  MoveL 2054 to (540.62, 2920.87, 513.19) mm, rotated rx -180 ry 0 rz -88.32 deg; joints [12.318, 40.901, 21.897, 21.013, -28.48, -28.65]
  MoveL 2055 to (543.06, 2922.34, 513.19) mm, rotated rx 180 ry 0 rz -88.32 deg; joints [12.364, 41.01, 22.057, 21.039, -28.543, -28.697]
  MoveL 2056 to (545.51, 2923.81, 513.19) mm, rotated rx -180 ry 0 rz -88.32 deg; joints [12.409, 41.12, 22.218, 21.064, -28.606, -28.743]
  MoveL 2057 to (547.96, 2925.26, 513.19) mm, rotated rx -180 ry 0 rz -88.32 deg; joints [12.455, 41.229, 22.379, 21.09, -28.67, -28.789]
  MoveL 2058 to (550.41, 2926.72, 513.19) mm, rotated rx 180 ry 0 rz -88.32 deg; joints [12.501, 41.339, 22.539, 21.115, -28.733, -28.835]
  MoveL 2059 to (552.87, 2928.16, 513.19) mm, rotated rx -180 ry 0 rz -88.32 deg; joints [12.547, 41.448, 22.7, 21.141, -28.797, -28.881]
  MoveL 2060 to (555.33, 2929.6, 513.19) mm, rotated rx -180 ry 0 rz -88.32 deg; joints [12.593, 41.558, 22.861, 21.166, -28.86, -28.926]
  MoveL 2061 to (557.79, 2931.02, 513.19) mm, rotated rx 180 ry 0 rz -88.32 deg; joints [12.639, 41.667, 23.021, 21.191, -28.924, -28.972]
  MoveL 2062 to (560.26, 2932.45, 513.19) mm, rotated rx 180 ry 0 rz -88.32 deg; joints [12.685, 41.776, 23.182, 21.216, -28.988, -29.018]
  MoveL 2063 to (562.74, 2933.86, 513.19) mm, rotated rx -180 ry 0 rz -88.32 deg; joints [12.731, 41.885, 23.343, 21.241, -29.052, -29.063]
  MoveL 2064 to (565.21, 2935.27, 513.19) mm, rotated rx -180 ry 0 rz -88.32 deg; joints [12.777, 41.995, 23.504, 21.266, -29.116, -29.108]
  MoveL 2065 to (567.69, 2936.67, 513.19) mm, rotated rx -180 ry 0 rz -88.32 deg; joints [12.823, 42.104, 23.665, 21.291, -29.18, -29.154]
  MoveL 2066 to (570.18, 2938.07, 513.19) mm, rotated rx 180 ry 0 rz -88.32 deg; joints [12.87, 42.213, 23.826, 21.316, -29.244, -29.199]
  MoveL 2067 to (572.67, 2939.46, 513.19) mm, rotated rx 180 ry 0 rz -88.32 deg; joints [12.916, 42.322, 23.987, 21.341, -29.309, -29.244]
  MoveL 2068 to (575.16, 2940.84, 513.19) mm, rotated rx 180 ry 0 rz -88.32 deg; joints [12.962, 42.431, 24.148, 21.366, -29.373, -29.289]
  MoveL 2069 to (577.66, 2942.21, 513.19) mm, rotated rx 180 ry 0 rz -88.32 deg; joints [13.009, 42.54, 24.31, 21.39, -29.438, -29.334]
  MoveL 2070 to (580.16, 2943.58, 513.19) mm, rotated rx 180 ry 0 rz -88.32 deg; joints [13.055, 42.649, 24.471, 21.415, -29.502, -29.378]
  MoveL 2071 to (582.66, 2944.94, 513.19) mm, rotated rx 180 ry 0 rz -88.32 deg; joints [13.102, 42.758, 24.632, 21.439, -29.567, -29.423]
  MoveL 2072 to (585.17, 2946.29, 513.19) mm, rotated rx 180 ry 0 rz -88.32 deg; joints [13.148, 42.867, 24.793, 21.463, -29.632, -29.468]
  MoveL 2073 to (587.68, 2947.64, 513.19) mm, rotated rx -180 ry 0 rz -88.32 deg; joints [13.195, 42.976, 24.955, 21.487, -29.697, -29.512]
  MoveL 2074 to (590.2, 2948.98, 513.19) mm, rotated rx -180 ry 0 rz -88.32 deg; joints [13.241, 43.085, 25.116, 21.512, -29.762, -29.557]
  MoveL 2075 to (592.72, 2950.31, 513.19) mm, rotated rx -180 ry 0 rz -88.32 deg; joints [13.288, 43.194, 25.278, 21.536, -29.828, -29.601]
  MoveL 2076 to (595.24, 2951.63, 513.19) mm, rotated rx -180 ry 0 rz -88.32 deg; joints [13.335, 43.303, 25.439, 21.56, -29.893, -29.645]
  MoveL 2077 to (597.77, 2952.95, 513.19) mm, rotated rx -180 ry 0 rz -88.32 deg; joints [13.382, 43.412, 25.601, 21.584, -29.959, -29.689]
  MoveL 2078 to (600.3, 2954.26, 513.19) mm, rotated rx 180 ry 0 rz -88.32 deg; joints [13.429, 43.521, 25.763, 21.607, -30.024, -29.733]
  MoveL 2079 to (602.83, 2955.57, 513.19) mm, rotated rx 180 ry 0 rz -88.32 deg; joints [13.475, 43.629, 25.924, 21.631, -30.09, -29.777]
  MoveL 2080 to (605.37, 2956.86, 513.19) mm, rotated rx 180 ry 0 rz -88.32 deg; joints [13.522, 43.738, 26.086, 21.655, -30.156, -29.821]
  MoveL 2081 to (607.91, 2958.15, 513.19) mm, rotated rx -180 ry 0 rz -88.32 deg; joints [13.569, 43.847, 26.248, 21.678, -30.222, -29.865]
  MoveL 2082 to (610.46, 2959.43, 513.19) mm, rotated rx -180 ry 0 rz -88.32 deg; joints [13.616, 43.955, 26.41, 21.702, -30.288, -29.908]
  MoveL 2083 to (613.01, 2960.71, 513.19) mm, rotated rx -180 ry 0 rz -88.32 deg; joints [13.663, 44.064, 26.572, 21.725, -30.354, -29.952]
  MoveL 2084 to (615.56, 2961.98, 513.19) mm, rotated rx 180 ry 0 rz -88.32 deg; joints [13.711, 44.173, 26.734, 21.749, -30.42, -29.996]
  MoveL 2085 to (618.11, 2963.24, 513.19) mm, rotated rx -180 ry 0 rz -88.32 deg; joints [13.758, 44.281, 26.896, 21.772, -30.486, -30.039]
  MoveL 2086 to (620.67, 2964.49, 513.19) mm, rotated rx 180 ry 0 rz -88.32 deg; joints [13.805, 44.39, 27.058, 21.795, -30.553, -30.082]
  MoveL 2087 to (623.24, 2965.74, 513.19) mm, rotated rx -180 ry 0 rz -88.32 deg; joints [13.852, 44.498, 27.22, 21.818, -30.619, -30.125]
  MoveL 2088 to (625.8, 2966.98, 513.19) mm, rotated rx -180 ry 0 rz -88.32 deg; joints [13.899, 44.607, 27.383, 21.841, -30.686, -30.168]
  MoveL 2089 to (628.37, 2968.21, 513.19) mm, rotated rx -180 ry 0 rz -88.32 deg; joints [13.947, 44.715, 27.545, 21.864, -30.753, -30.211]
  MoveL 2090 to (630.95, 2969.43, 513.19) mm, rotated rx -180 ry 0 rz -88.32 deg; joints [13.994, 44.824, 27.707, 21.887, -30.82, -30.254]
  MoveL 2091 to (633.52, 2970.65, 513.19) mm, rotated rx 180 ry 0 rz -88.32 deg; joints [14.042, 44.932, 27.87, 21.91, -30.887, -30.297]
  MoveL 2092 to (636.1, 2971.86, 513.19) mm, rotated rx -180 ry 0 rz -88.32 deg; joints [14.089, 45.041, 28.032, 21.933, -30.954, -30.34]
  MoveL 2093 to (638.69, 2973.06, 513.19) mm, rotated rx -180 ry 0 rz -88.32 deg; joints [14.137, 45.149, 28.195, 21.955, -31.021, -30.382]
  MoveL 2094 to (641.27, 2974.26, 513.19) mm, rotated rx 180 ry 0 rz -88.32 deg; joints [14.184, 45.257, 28.357, 21.978, -31.088, -30.425]
  MoveL 2095 to (643.86, 2975.45, 513.19) mm, rotated rx -180 ry 0 rz -88.32 deg; joints [14.232, 45.366, 28.52, 22, -31.156, -30.467]
  MoveL 2096 to (646.46, 2976.63, 513.19) mm, rotated rx 180 ry 0 rz -88.32 deg; joints [14.28, 45.474, 28.682, 22.023, -31.223, -30.51]
  MoveL 2097 to (649.05, 2977.8, 513.19) mm, rotated rx -180 ry 0 rz -88.32 deg; joints [14.327, 45.582, 28.845, 22.045, -31.291, -30.552]
  MoveL 2098 to (651.65, 2978.97, 513.19) mm, rotated rx -180 ry 0 rz -88.32 deg; joints [14.375, 45.691, 29.008, 22.067, -31.358, -30.594]
  MoveL 2099 to (654.26, 2980.13, 513.19) mm, rotated rx 180 ry 0 rz -88.32 deg; joints [14.423, 45.799, 29.171, 22.089, -31.426, -30.636]
  MoveL 2100 to (656.86, 2981.28, 513.19) mm, rotated rx 180 ry 0 rz -88.32 deg; joints [14.471, 45.907, 29.334, 22.112, -31.494, -30.678]
  MoveL 2101 to (659.47, 2982.43, 513.19) mm, rotated rx -180 ry 0 rz -88.32 deg; joints [14.518, 46.015, 29.497, 22.134, -31.562, -30.72]
  MoveL 2102 to (662.09, 2983.56, 513.19) mm, rotated rx -180 ry 0 rz -88.32 deg; joints [14.566, 46.124, 29.66, 22.156, -31.63, -30.762]
  MoveL 2103 to (664.7, 2984.69, 513.19) mm, rotated rx -180 ry 0 rz -88.32 deg; joints [14.614, 46.232, 29.823, 22.177, -31.699, -30.803]
  MoveL 2104 to (667.32, 2985.82, 513.19) mm, rotated rx 180 ry 0 rz -88.32 deg; joints [14.662, 46.34, 29.986, 22.199, -31.767, -30.845]
  MoveL 2105 to (669.95, 2986.93, 513.19) mm, rotated rx -180 ry 0 rz -88.32 deg; joints [14.71, 46.448, 30.149, 22.221, -31.835, -30.886]
  MoveL 2106 to (672.57, 2988.04, 513.19) mm, rotated rx 180 ry 0 rz -88.32 deg; joints [14.759, 46.556, 30.313, 22.243, -31.904, -30.928]
  MoveL 2107 to (675.2, 2989.14, 513.19) mm, rotated rx -180 ry 0 rz -88.32 deg; joints [14.807, 46.664, 30.476, 22.264, -31.973, -30.969]
  MoveL 2108 to (677.83, 2990.23, 513.19) mm, rotated rx -180 ry 0 rz -88.32 deg; joints [14.855, 46.772, 30.64, 22.286, -32.041, -31.01]
  MoveL 2109 to (680.47, 2991.32, 513.19) mm, rotated rx 180 ry 0 rz -88.32 deg; joints [14.903, 46.88, 30.803, 22.307, -32.11, -31.051]
  MoveL 2110 to (683.1, 2992.4, 513.19) mm, rotated rx 180 ry 0 rz -88.32 deg; joints [14.951, 46.988, 30.967, 22.329, -32.179, -31.092]
  MoveL 2111 to (685.75, 2993.47, 513.19) mm, rotated rx -180 ry 0 rz -88.32 deg; joints [15, 47.097, 31.13, 22.35, -32.248, -31.133]
  MoveL 2112 to (688.39, 2994.53, 513.19) mm, rotated rx 180 ry 0 rz -88.32 deg; joints [15.048, 47.205, 31.294, 22.371, -32.317, -31.174]
  MoveL 2113 to (691.04, 2995.59, 513.19) mm, rotated rx 180 ry 0 rz -88.32 deg; joints [15.096, 47.313, 31.458, 22.392, -32.387, -31.215]
  MoveL 2114 to (693.69, 2996.64, 513.19) mm, rotated rx -180 ry 0 rz -88.32 deg; joints [15.145, 47.421, 31.622, 22.413, -32.456, -31.255]
  MoveL 2115 to (696.34, 2997.68, 513.19) mm, rotated rx 180 ry 0 rz -88.32 deg; joints [15.193, 47.528, 31.786, 22.434, -32.526, -31.296]
  MoveL 2116 to (698.99, 2998.71, 513.19) mm, rotated rx 180 ry 0 rz -88.32 deg; joints [15.242, 47.636, 31.949, 22.455, -32.595, -31.336]
  MoveL 2117 to (701.65, 2999.74, 513.19) mm, rotated rx -180 ry 0 rz -88.32 deg; joints [15.29, 47.744, 32.114, 22.476, -32.665, -31.377]
  MoveL 2118 to (704.31, 3000.76, 513.19) mm, rotated rx -180 ry 0 rz -88.32 deg; joints [15.339, 47.852, 32.278, 22.497, -32.735, -31.417]
  MoveL 2119 to (706.98, 3001.77, 513.19) mm, rotated rx -180 ry 0 rz -88.32 deg; joints [15.387, 47.96, 32.442, 22.518, -32.805, -31.457]
  MoveL 2120 to (709.65, 3002.77, 513.19) mm, rotated rx -180 ry 0 rz -88.32 deg; joints [15.436, 48.068, 32.606, 22.538, -32.875, -31.497]
  MoveL 2121 to (712.32, 3003.77, 513.19) mm, rotated rx 180 ry 0 rz -88.32 deg; joints [15.485, 48.176, 32.77, 22.559, -32.945, -31.537]
  MoveL 2122 to (714.99, 3004.76, 513.19) mm, rotated rx 180 ry 0 rz -88.32 deg; joints [15.533, 48.284, 32.935, 22.58, -33.015, -31.577]
  MoveL 2123 to (717.66, 3005.74, 513.19) mm, rotated rx 180 ry 0 rz -88.32 deg; joints [15.582, 48.392, 33.099, 22.6, -33.085, -31.617]
  MoveL 2124 to (720.34, 3006.71, 513.19) mm, rotated rx -180 ry 0 rz -88.32 deg; joints [15.631, 48.5, 33.264, 22.62, -33.156, -31.656]
  MoveL 2125 to (723.02, 3007.68, 513.19) mm, rotated rx -180 ry 0 rz -88.32 deg; joints [15.68, 48.607, 33.428, 22.641, -33.226, -31.696]
  MoveL 2126 to (725.71, 3008.64, 513.19) mm, rotated rx 180 ry 0 rz -88.32 deg; joints [15.729, 48.715, 33.593, 22.661, -33.297, -31.735]
  MoveL 2127 to (728.39, 3009.59, 513.19) mm, rotated rx 180 ry 0 rz -88.32 deg; joints [15.778, 48.823, 33.758, 22.681, -33.368, -31.775]
  MoveL 2128 to (731.08, 3010.54, 513.19) mm, rotated rx -180 ry 0 rz -88.32 deg; joints [15.827, 48.931, 33.923, 22.701, -33.438, -31.814]
  MoveL 2129 to (733.77, 3011.47, 513.19) mm, rotated rx -180 ry 0 rz -88.32 deg; joints [15.876, 49.039, 34.087, 22.721, -33.509, -31.853]
  MoveL 2130 to (736.47, 3012.4, 513.19) mm, rotated rx 180 ry 0 rz -88.32 deg; joints [15.925, 49.147, 34.252, 22.741, -33.58, -31.892]
  MoveL 2131 to (739.16, 3013.32, 513.19) mm, rotated rx -180 ry 0 rz -88.32 deg; joints [15.974, 49.254, 34.417, 22.761, -33.651, -31.931]
  MoveL 2132 to (741.86, 3014.24, 513.19) mm, rotated rx -180 ry 0 rz -88.32 deg; joints [16.023, 49.362, 34.583, 22.781, -33.723, -31.97]
  MoveL 2133 to (744.57, 3015.14, 513.19) mm, rotated rx -180 ry 0 rz -88.32 deg; joints [16.072, 49.47, 34.748, 22.801, -33.794, -32.009]
  MoveL 2134 to (747.27, 3016.04, 513.19) mm, rotated rx 180 ry 0 rz -88.32 deg; joints [16.121, 49.578, 34.913, 22.821, -33.865, -32.048]
  MoveL 2135 to (749.98, 3016.93, 513.19) mm, rotated rx 180 ry 0 rz -88.32 deg; joints [16.17, 49.686, 35.078, 22.84, -33.937, -32.087]
  MoveL 2136 to (752.69, 3017.82, 513.19) mm, rotated rx -180 ry 0 rz -88.32 deg; joints [16.22, 49.793, 35.244, 22.86, -34.009, -32.125]
  MoveL 2137 to (755.4, 3018.69, 513.19) mm, rotated rx -180 ry 0 rz -88.32 deg; joints [16.269, 49.901, 35.409, 22.879, -34.08, -32.164]
  MoveL 2138 to (758.11, 3019.56, 513.19) mm, rotated rx -180 ry 0 rz -88.32 deg; joints [16.318, 50.009, 35.575, 22.899, -34.152, -32.202]
  MoveL 2139 to (760.83, 3020.42, 513.19) mm, rotated rx -180 ry 0 rz -88.32 deg; joints [16.368, 50.117, 35.741, 22.918, -34.224, -32.24]
  MoveL 2140 to (763.55, 3021.27, 513.19) mm, rotated rx 180 ry 0 rz -88.32 deg; joints [16.417, 50.224, 35.906, 22.937, -34.296, -32.278]
  MoveL 2141 to (766.27, 3022.12, 513.19) mm, rotated rx -180 ry 0 rz -88.32 deg; joints [16.466, 50.332, 36.072, 22.957, -34.368, -32.316]
  MoveL 2142 to (769, 3022.96, 513.19) mm, rotated rx -180 ry 0 rz -88.32 deg; joints [16.516, 50.44, 36.238, 22.976, -34.441, -32.354]
  MoveL 2143 to (771.72, 3023.79, 513.19) mm, rotated rx 180 ry 0 rz -88.32 deg; joints [16.565, 50.548, 36.404, 22.995, -34.513, -32.392]
  MoveL 2144 to (774.45, 3024.61, 513.19) mm, rotated rx -180 ry 0 rz -88.32 deg; joints [16.615, 50.655, 36.57, 23.014, -34.585, -32.43]
  MoveL 2145 to (777.18, 3025.42, 513.19) mm, rotated rx 180 ry 0 rz -88.32 deg; joints [16.665, 50.763, 36.736, 23.033, -34.658, -32.468]
  MoveL 2146 to (779.91, 3026.23, 513.19) mm, rotated rx 180 ry 0 rz -88.32 deg; joints [16.714, 50.871, 36.903, 23.052, -34.731, -32.505]
  MoveL 2147 to (782.65, 3027.03, 513.19) mm, rotated rx -180 ry 0 rz -88.32 deg; joints [16.764, 50.979, 37.069, 23.071, -34.803, -32.543]
  MoveL 2148 to (785.39, 3027.82, 513.19) mm, rotated rx -180 ry 0 rz -88.32 deg; joints [16.814, 51.086, 37.235, 23.09, -34.876, -32.58]
  MoveL 2149 to (788.13, 3028.61, 513.19) mm, rotated rx -180 ry 0 rz -88.32 deg; joints [16.863, 51.194, 37.402, 23.108, -34.949, -32.618]
  MoveL 2150 to (790.87, 3029.38, 513.19) mm, rotated rx -180 ry 0 rz -88.32 deg; joints [16.913, 51.302, 37.568, 23.127, -35.022, -32.655]
  MoveL 2151 to (793.61, 3030.15, 513.19) mm, rotated rx -180 ry 0 rz -88.32 deg; joints [16.963, 51.41, 37.735, 23.145, -35.095, -32.692]
  MoveL 2152 to (796.36, 3030.91, 513.19) mm, rotated rx 180 ry 0 rz -88.32 deg; joints [17.013, 51.518, 37.902, 23.164, -35.169, -32.729]
  MoveL 2153 to (799.11, 3031.66, 513.19) mm, rotated rx -180 ry 0 rz -88.32 deg; joints [17.062, 51.625, 38.069, 23.183, -35.242, -32.766]
  MoveL 2154 to (801.86, 3032.41, 513.19) mm, rotated rx -180 ry 0 rz -88.32 deg; joints [17.112, 51.733, 38.236, 23.201, -35.316, -32.803]
  MoveL 2155 to (804.61, 3033.15, 513.19) mm, rotated rx 180 ry 0 rz -88.32 deg; joints [17.162, 51.841, 38.403, 23.219, -35.389, -32.84]
  MoveL 2156 to (807.37, 3033.88, 513.19) mm, rotated rx 180 ry 0 rz -88.32 deg; joints [17.212, 51.949, 38.57, 23.238, -35.463, -32.876]
  MoveL 2157 to (810.12, 3034.6, 513.19) mm, rotated rx 180 ry 0 rz -88.32 deg; joints [17.262, 52.057, 38.737, 23.256, -35.537, -32.913]
  MoveL 2158 to (812.88, 3035.31, 513.19) mm, rotated rx -180 ry 0 rz -88.32 deg; joints [17.312, 52.164, 38.904, 23.274, -35.611, -32.949]
  MoveL 2159 to (815.64, 3036.02, 513.19) mm, rotated rx -180 ry 0 rz -88.32 deg; joints [17.362, 52.272, 39.072, 23.292, -35.685, -32.986]
  MoveL 2160 to (818.41, 3036.72, 513.19) mm, rotated rx 180 ry 0 rz -88.32 deg; joints [17.412, 52.38, 39.239, 23.31, -35.759, -33.022]
  MoveL 2161 to (821.17, 3037.41, 513.19) mm, rotated rx 180 ry 0 rz -88.32 deg; joints [17.462, 52.488, 39.407, 23.328, -35.833, -33.058]
  MoveL 2162 to (823.94, 3038.1, 513.19) mm, rotated rx -180 ry 0 rz -88.32 deg; joints [17.513, 52.596, 39.575, 23.346, -35.907, -33.094]
  MoveL 2163 to (826.71, 3038.77, 513.19) mm, rotated rx -180 ry 0 rz -88.32 deg; joints [17.563, 52.704, 39.743, 23.364, -35.982, -33.13]
  MoveL 2164 to (829.48, 3039.44, 513.19) mm, rotated rx 180 ry 0 rz -88.32 deg; joints [17.613, 52.812, 39.911, 23.382, -36.056, -33.166]
  MoveL 2165 to (832.25, 3040.1, 513.19) mm, rotated rx 180 ry 0 rz -88.32 deg; joints [17.663, 52.919, 40.079, 23.399, -36.131, -33.202]
  MoveL 2166 to (835.02, 3040.75, 513.19) mm, rotated rx -180 ry 0 rz -88.32 deg; joints [17.714, 53.027, 40.247, 23.417, -36.206, -33.238]
  MoveL 2167 to (837.8, 3041.4, 513.19) mm, rotated rx 180 ry 0 rz -88.32 deg; joints [17.764, 53.135, 40.415, 23.435, -36.28, -33.273]
  MoveL 2168 to (840.58, 3042.03, 513.19) mm, rotated rx 180 ry 0 rz -88.32 deg; joints [17.814, 53.243, 40.583, 23.452, -36.355, -33.309]
  MoveL 2169 to (843.36, 3042.66, 513.19) mm, rotated rx -180 ry 0 rz -88.32 deg; joints [17.865, 53.351, 40.752, 23.47, -36.43, -33.344]
  MoveL 2170 to (846.14, 3043.28, 513.19) mm, rotated rx 180 ry 0 rz -88.32 deg; joints [17.915, 53.459, 40.92, 23.487, -36.506, -33.379]
  MoveL 2171 to (848.92, 3043.9, 513.19) mm, rotated rx -180 ry 0 rz -88.32 deg; joints [17.965, 53.567, 41.089, 23.505, -36.581, -33.415]
  MoveL 2172 to (851.7, 3044.5, 513.19) mm, rotated rx -180 ry 0 rz -88.32 deg; joints [18.016, 53.675, 41.258, 23.522, -36.656, -33.45]
  MoveL 2173 to (854.49, 3045.1, 513.19) mm, rotated rx 180 ry 0 rz -88.32 deg; joints [18.066, 53.783, 41.427, 23.539, -36.732, -33.485]
  MoveL 2174 to (857.28, 3045.69, 513.19) mm, rotated rx 180 ry 0 rz -88.32 deg; joints [18.117, 53.891, 41.596, 23.556, -36.807, -33.52]
  MoveL 2175 to (860.07, 3046.27, 513.19) mm, rotated rx -180 ry 0 rz -88.32 deg; joints [18.167, 54, 41.765, 23.573, -36.883, -33.555]
  MoveL 2176 to (862.86, 3046.85, 513.19) mm, rotated rx 180 ry 0 rz -88.32 deg; joints [18.218, 54.108, 41.934, 23.59, -36.959, -33.589]
  MoveL 2177 to (865.65, 3047.42, 513.19) mm, rotated rx 180 ry 0 rz -88.32 deg; joints [18.269, 54.216, 42.103, 23.607, -37.035, -33.624]
  MoveL 2178 to (868.45, 3047.97, 513.19) mm, rotated rx -180 ry 0 rz -88.32 deg; joints [18.319, 54.324, 42.273, 23.624, -37.111, -33.659]
  MoveL 2179 to (871.24, 3048.53, 513.19) mm, rotated rx 180 ry 0 rz -88.32 deg; joints [18.37, 54.432, 42.442, 23.641, -37.187, -33.693]
  MoveL 2180 to (874.04, 3049.07, 513.19) mm, rotated rx 180 ry 0 rz -88.32 deg; joints [18.421, 54.54, 42.612, 23.658, -37.263, -33.727]
  MoveL 2181 to (876.84, 3049.6, 513.19) mm, rotated rx 180 ry 0 rz -88.32 deg; joints [18.471, 54.649, 42.782, 23.675, -37.339, -33.762]
  MoveL 2182 to (879.64, 3050.13, 513.19) mm, rotated rx 180 ry 0 rz -88.32 deg; joints [18.522, 54.757, 42.952, 23.692, -37.416, -33.796]
  MoveL 2183 to (882.44, 3050.65, 513.19) mm, rotated rx 180 ry 0 rz -88.32 deg; joints [18.573, 54.865, 43.122, 23.708, -37.492, -33.83]
  MoveL 2184 to (885.25, 3051.16, 513.19) mm, rotated rx -180 ry 0 rz -88.32 deg; joints [18.624, 54.974, 43.292, 23.725, -37.569, -33.864]
  MoveL 2185 to (888.05, 3051.67, 513.19) mm, rotated rx 180 ry 0 rz -88.32 deg; joints [18.675, 55.082, 43.463, 23.741, -37.646, -33.897]
  MoveL 2186 to (890.86, 3052.16, 513.19) mm, rotated rx 180 ry 0 rz -88.32 deg; joints [18.726, 55.19, 43.633, 23.758, -37.723, -33.931]
  MoveL 2187 to (893.67, 3052.65, 513.19) mm, rotated rx -180 ry 0 rz -88.32 deg; joints [18.776, 55.299, 43.804, 23.774, -37.8, -33.965]
  MoveL 2188 to (896.48, 3053.13, 513.19) mm, rotated rx 180 ry 0 rz -88.32 deg; joints [18.827, 55.407, 43.974, 23.791, -37.877, -33.998]
  MoveL 2189 to (899.29, 3053.6, 513.19) mm, rotated rx -180 ry 0 rz -88.32 deg; joints [18.878, 55.516, 44.145, 23.807, -37.954, -34.032]
  MoveL 2190 to (902.1, 3054.07, 513.19) mm, rotated rx -180 ry 0 rz -88.32 deg; joints [18.929, 55.624, 44.316, 23.823, -38.031, -34.065]
  MoveL 2191 to (904.91, 3054.52, 513.19) mm, rotated rx -180 ry 0 rz -88.32 deg; joints [18.98, 55.733, 44.487, 23.839, -38.109, -34.098]
  MoveL 2192 to (907.72, 3054.97, 513.19) mm, rotated rx 180 ry 0 rz -88.32 deg; joints [19.031, 55.842, 44.659, 23.856, -38.186, -34.132]
  MoveL 2193 to (910.54, 3055.41, 513.19) mm, rotated rx -180 ry 0 rz -88.32 deg; joints [19.082, 55.95, 44.83, 23.872, -38.264, -34.165]
  MoveL 2194 to (913.36, 3055.85, 513.19) mm, rotated rx -180 ry 0 rz -88.32 deg; joints [19.134, 56.059, 45.002, 23.888, -38.342, -34.198]
  MoveL 2195 to (916.18, 3056.27, 513.19) mm, rotated rx 180 ry 0 rz -88.32 deg; joints [19.185, 56.168, 45.173, 23.904, -38.419, -34.23]
  MoveL 2196 to (918.99, 3056.69, 513.19) mm, rotated rx -180 ry 0 rz -88.32 deg; joints [19.236, 56.276, 45.345, 23.92, -38.497, -34.263]
  MoveL 2197 to (921.81, 3057.1, 513.19) mm, rotated rx 180 ry 0 rz -88.32 deg; joints [19.287, 56.385, 45.517, 23.935, -38.576, -34.296]
  MoveL 2198 to (924.64, 3057.5, 513.19) mm, rotated rx -180 ry 0 rz -88.32 deg; joints [19.338, 56.494, 45.689, 23.951, -38.654, -34.328]
  MoveL 2199 to (927.46, 3057.89, 513.19) mm, rotated rx -180 ry 0 rz -88.32 deg; joints [19.39, 56.603, 45.862, 23.967, -38.732, -34.361]
  MoveL 2200 to (930.28, 3058.28, 513.19) mm, rotated rx -180 ry 0 rz -88.32 deg; joints [19.441, 56.712, 46.034, 23.983, -38.811, -34.393]
  MoveL 2201 to (933.11, 3058.65, 513.19) mm, rotated rx -180 ry 0 rz -88.32 deg; joints [19.492, 56.821, 46.207, 23.998, -38.889, -34.425]
  MoveL 2202 to (935.93, 3059.02, 513.19) mm, rotated rx -180 ry 0 rz -88.32 deg; joints [19.543, 56.93, 46.379, 24.014, -38.968, -34.457]
  MoveL 2203 to (938.76, 3059.39, 513.19) mm, rotated rx -180 ry 0 rz -88.32 deg; joints [19.595, 57.039, 46.552, 24.029, -39.047, -34.489]
  MoveL 2204 to (941.59, 3059.74, 513.19) mm, rotated rx -180 ry 0 rz -88.32 deg; joints [19.646, 57.149, 46.725, 24.045, -39.126, -34.521]
  MoveL 2205 to (944.42, 3060.09, 513.19) mm, rotated rx 180 ry 0 rz -88.32 deg; joints [19.698, 57.258, 46.899, 24.06, -39.205, -34.553]
  MoveL 2206 to (947.25, 3060.42, 513.19) mm, rotated rx -180 ry 0 rz -88.32 deg; joints [19.749, 57.367, 47.072, 24.075, -39.284, -34.585]
  MoveL 2207 to (950.08, 3060.75, 513.19) mm, rotated rx -180 ry 0 rz -88.32 deg; joints [19.8, 57.477, 47.246, 24.091, -39.363, -34.616]
  MoveL 2208 to (952.91, 3061.07, 513.19) mm, rotated rx 180 ry 0 rz -88.32 deg; joints [19.852, 57.586, 47.42, 24.106, -39.443, -34.648]
  MoveL 2209 to (955.74, 3061.39, 513.19) mm, rotated rx -180 ry 0 rz -88.32 deg; joints [19.903, 57.695, 47.593, 24.121, -39.522, -34.679]
  MoveL 2210 to (958.57, 3061.7, 513.19) mm, rotated rx -180 ry 0 rz -88.32 deg; joints [19.955, 57.805, 47.768, 24.136, -39.602, -34.71]
  MoveL 2211 to (961.41, 3061.99, 513.19) mm, rotated rx 180 ry 0 rz -88.32 deg; joints [20.006, 57.915, 47.942, 24.151, -39.682, -34.742]
  MoveL 2212 to (964.24, 3062.28, 513.19) mm, rotated rx 180 ry 0 rz -88.32 deg; joints [20.058, 58.024, 48.116, 24.166, -39.762, -34.773]
  MoveL 2213 to (967.08, 3062.57, 513.19) mm, rotated rx -180 ry 0 rz -88.32 deg; joints [20.11, 58.134, 48.291, 24.181, -39.842, -34.804]
  MoveL 2214 to (969.92, 3062.84, 513.19) mm, rotated rx -180 ry 0 rz -88.32 deg; joints [20.161, 58.244, 48.466, 24.196, -39.922, -34.834]
  MoveL 2215 to (972.75, 3063.11, 513.19) mm, rotated rx 180 ry 0 rz -88.32 deg; joints [20.213, 58.354, 48.641, 24.211, -40.002, -34.865]
  MoveL 2216 to (975.59, 3063.36, 513.19) mm, rotated rx 180 ry 0 rz -88.32 deg; joints [20.265, 58.464, 48.816, 24.225, -40.082, -34.896]
  MoveL 2217 to (978.43, 3063.61, 513.19) mm, rotated rx -180 ry 0 rz -88.32 deg; joints [20.316, 58.574, 48.992, 24.24, -40.163, -34.926]
  MoveL 2218 to (981.27, 3063.86, 513.19) mm, rotated rx -180 ry 0 rz -88.32 deg; joints [20.368, 58.684, 49.167, 24.255, -40.244, -34.957]
  MoveL 2219 to (984.11, 3064.09, 513.19) mm, rotated rx -180 ry 0 rz -88.32 deg; joints [20.42, 58.794, 49.343, 24.269, -40.324, -34.987]
  MoveL 2220 to (986.95, 3064.32, 513.19) mm, rotated rx 180 ry 0 rz -88.32 deg; joints [20.472, 58.904, 49.519, 24.284, -40.405, -35.017]
  MoveL 2221 to (989.79, 3064.54, 513.19) mm, rotated rx -180 ry 0 rz -88.32 deg; joints [20.523, 59.015, 49.695, 24.298, -40.486, -35.047]
  MoveL 2222 to (992.63, 3064.75, 513.19) mm, rotated rx 180 ry 0 rz -88.32 deg; joints [20.575, 59.125, 49.872, 24.313, -40.568, -35.077]
  MoveL 2223 to (995.48, 3064.95, 513.19) mm, rotated rx -180 ry 0 rz -88.32 deg; joints [20.627, 59.236, 50.049, 24.327, -40.649, -35.107]
  MoveL 2224 to (998.32, 3065.14, 513.19) mm, rotated rx 180 ry 0 rz -88.32 deg; joints [20.679, 59.347, 50.225, 24.341, -40.73, -35.136]
  MoveL 2225 to (1001.16, 3065.33, 513.19) mm, rotated rx -180 ry 0 rz -88.32 deg; joints [20.731, 59.457, 50.403, 24.355, -40.812, -35.166]
  MoveL 2226 to (1004.01, 3065.51, 513.19) mm, rotated rx 180 ry 0 rz -88.32 deg; joints [20.783, 59.568, 50.58, 24.37, -40.894, -35.196]
  MoveL 2227 to (1006.85, 3065.68, 513.19) mm, rotated rx -180 ry 0 rz -88.32 deg; joints [20.835, 59.679, 50.757, 24.384, -40.976, -35.225]
  MoveL 2228 to (1009.7, 3065.84, 513.19) mm, rotated rx 180 ry 0 rz -88.32 deg; joints [20.887, 59.79, 50.935, 24.398, -41.058, -35.254]
  MoveL 2229 to (1012.54, 3066, 513.19) mm, rotated rx -180 ry 0 rz -88.32 deg; joints [20.939, 59.901, 51.113, 24.412, -41.14, -35.283]
  MoveL 2230 to (1015.39, 3066.14, 513.19) mm, rotated rx -180 ry 0 rz -88.32 deg; joints [20.991, 60.012, 51.292, 24.426, -41.222, -35.312]
  MoveL 2231 to (1018.24, 3066.28, 513.19) mm, rotated rx -180 ry 0 rz -88.32 deg; joints [21.043, 60.124, 51.47, 24.439, -41.305, -35.341]
  MoveL 2232 to (1021.08, 3066.41, 513.19) mm, rotated rx -180 ry 0 rz -88.32 deg; joints [21.095, 60.235, 51.649, 24.453, -41.387, -35.37]
  MoveL 2233 to (1023.93, 3066.54, 513.19) mm, rotated rx 180 ry 0 rz -88.32 deg; joints [21.147, 60.347, 51.828, 24.467, -41.47, -35.398]
  MoveL 2234 to (1026.78, 3066.65, 513.19) mm, rotated rx -180 ry 0 rz -88.32 deg; joints [21.199, 60.458, 52.007, 24.481, -41.553, -35.427]
  MoveL 2235 to (1029.63, 3066.76, 513.19) mm, rotated rx -180 ry 0 rz -88.32 deg; joints [21.251, 60.57, 52.187, 24.494, -41.636, -35.455]
  MoveL 2236 to (1032.47, 3066.86, 513.19) mm, rotated rx -180 ry 0 rz -88.32 deg; joints [21.303, 60.682, 52.367, 24.508, -41.719, -35.484]
  MoveL 2237 to (1035.32, 3066.95, 513.19) mm, rotated rx -180 ry 0 rz -88.32 deg; joints [21.355, 60.794, 52.547, 24.521, -41.802, -35.512]
  MoveL 2238 to (1038.17, 3067.03, 513.19) mm, rotated rx 180 ry 0 rz -88.32 deg; joints [21.407, 60.906, 52.727, 24.535, -41.886, -35.54]
  MoveL 2239 to (1041.02, 3067.11, 513.19) mm, rotated rx -180 ry 0 rz -88.32 deg; joints [21.46, 61.019, 52.908, 24.548, -41.969, -35.568]
  MoveL 2240 to (1043.87, 3067.17, 513.19) mm, rotated rx -180 ry 0 rz -88.32 deg; joints [21.512, 61.131, 53.089, 24.561, -42.053, -35.595]
  MoveL 2241 to (1046.72, 3067.23, 513.19) mm, rotated rx 180 ry 0 rz -88.32 deg; joints [21.564, 61.244, 53.27, 24.574, -42.137, -35.623]
  MoveL 2242 to (1049.57, 3067.28, 513.19) mm, rotated rx -180 ry 0 rz -88.32 deg; joints [21.616, 61.356, 53.451, 24.587, -42.221, -35.65]
  MoveL 2243 to (1052.42, 3067.32, 513.19) mm, rotated rx -180 ry 0 rz -88.32 deg; joints [21.669, 61.469, 53.633, 24.601, -42.306, -35.678]
  MoveL 2244 to (1055.27, 3067.36, 513.19) mm, rotated rx -180 ry 0 rz -88.32 deg; joints [21.721, 61.582, 53.815, 24.614, -42.39, -35.705]
  MoveL 2245 to (1058.12, 3067.39, 513.19) mm, rotated rx -180 ry 0 rz -88.32 deg; joints [21.773, 61.695, 53.998, 24.627, -42.475, -35.732]
  MoveL 2246 to (1060.97, 3067.41, 513.19) mm, rotated rx -180 ry 0 rz -88.32 deg; joints [21.826, 61.808, 54.18, 24.639, -42.56, -35.759]
  MoveL 2247 to (1063.82, 3067.42, 513.19) mm, rotated rx 180 ry 0 rz -88.32 deg; joints [21.878, 61.922, 54.364, 24.652, -42.644, -35.786]
  MoveL 2248 to (1066.67, 3067.42, 513.19) mm, rotated rx 180 ry 0 rz -88.32 deg; joints [21.931, 62.035, 54.547, 24.665, -42.73, -35.812]
  MoveL 2249 to (1069.52, 3067.41, 513.19) mm, rotated rx -180 ry 0 rz -88.32 deg; joints [21.983, 62.149, 54.731, 24.678, -42.815, -35.839]
  MoveL 2250 to (1072.37, 3067.4, 513.19) mm, rotated rx -180 ry 0 rz -88.32 deg; joints [22.035, 62.263, 54.915, 24.69, -42.9, -35.865]
  MoveL 2251 to (1075.22, 3067.38, 513.19) mm, rotated rx -180 ry 0 rz -88.32 deg; joints [22.088, 62.377, 55.099, 24.703, -42.986, -35.892]
  Set speed (100.0 mm/s)
  MoveL 2252 to (1075.22, 3067.38, 556.29) mm, rotated rx -180 ry 0 rz -88.32 deg; joints [22.088, 62.498, 56.778, 24.03, -44.405, -34.961]
  MoveL 2253 to (416.69, 1842.51, 556.29) mm, rotated rx -180 ry 0 rz -88.32 deg; joints [16.434, -12.998, -39.492, 33.424, -23.517, -44.201]
  Set speed (5.6 mm/s)
  MoveL 2254 to (416.69, 1842.51, 552.29) mm, rotated rx 180 ry 0 rz -88.32 deg; joints [16.434, -12.924, -39.576, 33.624, -23.386, -44.42]
  MoveL 2255 to (416.69, 1842.51, 532.29) mm, rotated rx -180 ry 0 rz -88.32 deg; joints [16.434, -12.543, -39.985, 34.666, -22.732, -45.552]
  Set speed (91.9 mm/s)
  MoveL 2256 to (364.31, 1842.97, 532.29) mm, rotated rx -180 ry 0 rz -88.32 deg; joints [14.515, -13.29, -40.608, 31.913, -21.899, -41.623]
  MoveL 2257 to (364.3, 1842.96, 532.29) mm, rotated rx -180 ry 0 rz -88.32 deg; joints [14.515, -13.29, -40.608, 31.913, -21.9, -41.623]
  MoveL 2258 to (363.38, 1738.2, 532.29) mm, rotated rx -180 ry 0 rz -88.32 deg; joints [15.551, -19.08, -45.212, 31.828, -23.396, -42.036]
  MoveL 2259 to (468.15, 1737.27, 532.29) mm, rotated rx -180 ry 0 rz -88.32 deg; joints [19.596, -17.284, -43.827, 37.188, -25.115, -49.88]
  MoveL 2260 to (468.15, 1737.28, 532.29) mm, rotated rx -180 ry 0 rz -88.32 deg; joints [19.596, -17.284, -43.827, 37.188, -25.115, -49.88]
  MoveL 2261 to (469.08, 1842.04, 532.29) mm, rotated rx -180 ry 0 rz -88.32 deg; joints [18.316, -11.712, -39.282, 37.134, -23.607, -49.182]
  MoveL 2262 to (416.69, 1842.51, 532.29) mm, rotated rx -180 ry 0 rz -88.32 deg; joints [16.434, -12.543, -39.985, 34.666, -22.732, -45.552]
  Set speed (5.6 mm/s)
  MoveL 2263 to (416.69, 1842.51, 513.19) mm, rotated rx -180 ry 0 rz -88.32 deg; joints [16.434, -12.164, -40.364, 35.725, -22.112, -46.698]
  Set speed (91.9 mm/s)
  MoveL 2264 to (364.31, 1842.97, 513.19) mm, rotated rx -180 ry 0 rz -88.32 deg; joints [14.515, -12.91, -40.99, 32.946, -21.257, -42.733]
  MoveL 2265 to (364.3, 1842.96, 513.19) mm, rotated rx 180 ry 0 rz -88.32 deg; joints [14.515, -12.91, -40.99, 32.946, -21.257, -42.733]
  MoveL 2266 to (363.38, 1738.2, 513.19) mm, rotated rx -180 ry 0 rz -88.32 deg; joints [15.551, -18.701, -45.616, 32.812, -22.734, -43.104]
  MoveL 2267 to (468.15, 1737.27, 513.19) mm, rotated rx -180 ry 0 rz -88.32 deg; joints [19.596, -16.904, -44.224, 38.216, -24.5, -51.012]
  MoveL 2268 to (468.15, 1737.28, 513.19) mm, rotated rx -180 ry 0 rz -88.32 deg; joints [19.596, -16.904, -44.224, 38.216, -24.5, -51.012]
  MoveL 2269 to (469.08, 1842.04, 513.19) mm, rotated rx -180 ry 0 rz -88.32 deg; joints [18.316, -11.333, -39.659, 38.205, -23.009, -50.348]
  MoveL 2270 to (416.69, 1842.51, 513.19) mm, rotated rx -180 ry 0 rz -88.32 deg; joints [16.434, -12.164, -40.364, 35.725, -22.112, -46.698]
  Set speed (100.0 mm/s)
  MoveL 2271 to (416.69, 1842.51, 556.29) mm, rotated rx -180 ry 0 rz -88.32 deg; joints [16.434, -12.998, -39.492, 33.424, -23.517, -44.201]
  MoveL 2272 to (915.55, 1522.51, 556.29) mm, rotated rx 180 ry 0 rz -88.32 deg; joints [39.249, -15.841, -41.816, 49.069, -37.815, -73.844]
  Set speed (5.6 mm/s)
  MoveL 2273 to (915.55, 1522.51, 552.29) mm, rotated rx 180 ry 0 rz -88.32 deg; joints [39.249, -15.767, -41.901, 49.225, -37.71, -74.041]
  MoveL 2274 to (915.55, 1522.51, 532.29) mm, rotated rx -180 ry 0 rz -88.32 deg; joints [39.249, -15.386, -42.321, 50.021, -37.191, -75.044]
  Set speed (91.9 mm/s)
  MoveL 2275 to (915.67, 1535.21, 532.29) mm, rotated rx -180 ry 0 rz -88.32 deg; joints [38.94, -14.826, -41.869, 50.036, -36.912, -74.888]
  MoveL 2276 to (916.27, 1603.78, 532.29) mm, rotated rx -180 ry 0 rz -88.32 deg; joints [37.346, -11.818, -39.373, 50.06, -35.497, -74.011]
  Set speed (100.0 mm/s)
  MoveL 2277 to (916.27, 1603.78, 556.29) mm, rotated rx -180 ry 0 rz -88.32 deg; joints [37.346, -12.273, -38.884, 49.064, -36.109, -72.783]
  MoveL 2278 to (996.89, 1528.14, 556.29) mm, rotated rx -180 ry 0 rz -88.32 deg; joints [41.483, -12.67, -39.217, 50.268, -38.971, -76.634]
  Set speed (5.6 mm/s)
  MoveL 2279 to (996.89, 1528.14, 552.29) mm, rotated rx -180 ry 0 rz -88.32 deg; joints [41.483, -12.595, -39.3, 50.418, -38.871, -76.827]
  MoveL 2280 to (996.89, 1528.14, 532.29) mm, rotated rx -180 ry 0 rz -88.32 deg; joints [41.483, -12.215, -39.708, 51.182, -38.373, -77.806]
  Set speed (91.9 mm/s)
  MoveL 2281 to (928.31, 1528.74, 532.29) mm, rotated rx -180 ry 0 rz -88.32 deg; joints [39.478, -14.658, -41.732, 50.23, -37.259, -75.437]
  Set speed (100.0 mm/s)
  MoveL 2282 to (928.31, 1528.74, 556.29) mm, rotated rx -180 ry 0 rz -88.32 deg; joints [39.478, -15.113, -41.23, 49.28, -37.878, -74.239]
  MoveL 2283 to (915.55, 1522.51, 556.29) mm, rotated rx 180 ry 0 rz -88.32 deg; joints [39.249, -15.841, -41.816, 49.069, -37.815, -73.844]
  Set speed (5.6 mm/s)
  MoveL 2284 to (915.55, 1522.51, 533.29) mm, rotated rx 180 ry 0 rz -88.32 deg; joints [39.249, -15.405, -42.3, 49.981, -37.217, -74.993]
  MoveL 2285 to (915.55, 1522.51, 513.19) mm, rotated rx -180 ry 0 rz -88.32 deg; joints [39.249, -15.005, -42.711, 50.81, -36.701, -76.031]
  Set speed (91.9 mm/s)
  MoveL 2286 to (915.67, 1535.21, 513.19) mm, rotated rx -180 ry 0 rz -88.32 deg; joints [38.94, -14.445, -42.256, 50.831, -36.423, -75.879]
  MoveL 2287 to (916.27, 1603.78, 513.19) mm, rotated rx -180 ry 0 rz -88.32 deg; joints [37.346, -11.44, -39.75, 50.885, -35.016, -75.021]
  Set speed (100.0 mm/s)
  MoveL 2288 to (916.27, 1603.78, 556.29) mm, rotated rx -180 ry 0 rz -88.32 deg; joints [37.346, -12.273, -38.884, 49.064, -36.109, -72.783]
  MoveL 2289 to (996.89, 1528.14, 556.29) mm, rotated rx -180 ry 0 rz -88.32 deg; joints [41.483, -12.67, -39.217, 50.268, -38.971, -76.634]
  Set speed (5.6 mm/s)
  MoveL 2290 to (996.89, 1528.14, 533.29) mm, rotated rx -180 ry 0 rz -88.32 deg; joints [41.483, -12.234, -39.688, 51.144, -38.398, -77.756]
  MoveL 2291 to (996.89, 1528.14, 513.19) mm, rotated rx -180 ry 0 rz -88.32 deg; joints [41.483, -11.836, -40.086, 51.938, -37.902, -78.766]
  Set speed (91.9 mm/s)
  MoveL 2292 to (928.31, 1528.74, 513.19) mm, rotated rx -180 ry 0 rz -88.32 deg; joints [39.478, -14.278, -42.119, 51.016, -36.773, -76.422]
  Set speed (100.0 mm/s)
  MoveL 2293 to (928.31, 1528.74, 556.29) mm, rotated rx -180 ry 0 rz -88.32 deg; joints [39.478, -15.113, -41.23, 49.28, -37.878, -74.239]
  MoveL 2294 to (708.17, 1429.08, 556.29) mm, rotated rx -180 ry 0 rz -88.32 deg; joints [34.658, -27.904, -50.623, 44.105, -37.011, -65.215]
  Set speed (5.6 mm/s)
  MoveL 2295 to (708.17, 1429.08, 552.29) mm, rotated rx -180 ry 0 rz -88.32 deg; joints [34.658, -27.835, -50.719, 44.258, -36.892, -65.407]
  MoveL 2296 to (708.17, 1429.08, 532.29) mm, rotated rx -180 ry 0 rz -88.32 deg; joints [34.658, -27.477, -51.194, 45.047, -36.299, -66.39]
  Set speed (91.9 mm/s)
  MoveL 2297 to (789.45, 1428.36, 532.29) mm, rotated rx -180 ry 0 rz -88.32 deg; joints [37.589, -24.445, -49.125, 47.234, -37.561, -70.629]
  Set speed (100.0 mm/s)
  MoveL 2298 to (789.45, 1428.36, 556.29) mm, rotated rx -180 ry 0 rz -88.32 deg; joints [37.589, -24.884, -48.571, 46.305, -38.241, -69.451]
  MoveL 2299 to (708.17, 1429.08, 556.29) mm, rotated rx -180 ry 0 rz -88.32 deg; joints [34.658, -27.904, -50.623, 44.105, -37.011, -65.215]
  Set speed (5.6 mm/s)
  MoveL 2300 to (708.17, 1429.08, 533.29) mm, rotated rx 180 ry 0 rz -88.32 deg; joints [34.658, -27.496, -51.171, 45.007, -36.329, -66.34]
  MoveL 2301 to (708.17, 1429.08, 513.19) mm, rotated rx -180 ry 0 rz -88.32 deg; joints [34.658, -27.115, -51.637, 45.835, -35.735, -67.364]
  Set speed (91.9 mm/s)
  MoveL 2302 to (789.45, 1428.36, 513.19) mm, rotated rx 180 ry 0 rz -88.32 deg; joints [37.589, -24.074, -49.553, 48.009, -37.023, -71.602]
  Set speed (100.0 mm/s)
  MoveL 2303 to (789.45, 1428.36, 556.29) mm, rotated rx -180 ry 0 rz -88.32 deg; joints [37.589, -24.884, -48.571, 46.305, -38.241, -69.451]
  MoveL 2304 to (922.45, 2304.8, 556.29) mm, rotated rx -180 ry 0 rz -88.32 deg; joints [25.988, 17.43, -8.212, 41.857, -29.472, -58.291]
  Set speed (5.6 mm/s)
  MoveL 2305 to (922.45, 2304.8, 552.29) mm, rotated rx -180 ry 0 rz -88.32 deg; joints [25.988, 17.491, -8.282, 42.013, -29.375, -58.47]
  MoveL 2306 to (922.45, 2304.8, 532.29) mm, rotated rx -180 ry 0 rz -88.32 deg; joints [25.988, 17.799, -8.63, 42.806, -28.891, -59.378]
  Set speed (91.9 mm/s)
  MoveL 2307 to (923.05, 2373.37, 532.29) mm, rotated rx -180 ry 0 rz -88.32 deg; joints [25.219, 20.714, -5.01, 41.361, -28.95, -57.341]
  MoveL 2308 to (923.16, 2386.07, 532.29) mm, rotated rx -180 ry 0 rz -88.32 deg; joints [25.081, 21.258, -4.323, 41.082, -28.976, -56.954]
  Set speed (100.0 mm/s)
  MoveL 2309 to (923.16, 2386.07, 556.29) mm, rotated rx -180 ry 0 rz -88.32 deg; joints [25.081, 20.906, -3.904, 40.185, -29.561, -55.926]
  MoveL 2310 to (935.81, 2379.6, 556.29) mm, rotated rx 180 ry 0 rz -88.32 deg; joints [25.449, 20.885, -3.931, 40.484, -29.774, -56.448]
  Set speed (5.6 mm/s)
  MoveL 2311 to (935.81, 2379.6, 552.29) mm, rotated rx 180 ry 0 rz -88.32 deg; joints [25.449, 20.942, -4.002, 40.631, -29.676, -56.617]
  MoveL 2312 to (935.81, 2379.6, 532.29) mm, rotated rx -180 ry 0 rz -88.32 deg; joints [25.449, 21.237, -4.35, 41.379, -29.19, -57.476]
  Set speed (91.9 mm/s)
  MoveL 2313 to (1004.39, 2379, 532.29) mm, rotated rx -180 ry 0 rz -88.32 deg; joints [27.042, 22.645, -2.558, 42.123, -30.435, -59.12]
  Set speed (100.0 mm/s)
  MoveL 2314 to (1004.39, 2379, 556.29) mm, rotated rx -180 ry 0 rz -88.32 deg; joints [27.042, 22.299, -2.138, 41.265, -31.007, -58.122]
  MoveL 2315 to (935.81, 2379.6, 556.29) mm, rotated rx 180 ry 0 rz -88.32 deg; joints [25.449, 20.885, -3.931, 40.484, -29.774, -56.448]
  Set speed (5.6 mm/s)
  MoveL 2316 to (935.81, 2379.6, 533.29) mm, rotated rx -180 ry 0 rz -88.32 deg; joints [25.449, 21.222, -4.333, 41.341, -29.214, -57.432]
  MoveL 2317 to (935.81, 2379.6, 513.19) mm, rotated rx -180 ry 0 rz -88.32 deg; joints [25.449, 21.529, -4.671, 42.116, -28.733, -58.318]
  Set speed (91.9 mm/s)
  MoveL 2318 to (1004.39, 2379, 513.19) mm, rotated rx -180 ry 0 rz -88.32 deg; joints [27.042, 22.931, -2.88, 42.828, -29.986, -59.936]
  Set speed (100.0 mm/s)
  MoveL 2319 to (1004.39, 2379, 556.29) mm, rotated rx -180 ry 0 rz -88.32 deg; joints [27.042, 22.299, -2.138, 41.265, -31.007, -58.122]
  MoveL 2320 to (922.45, 2304.8, 556.29) mm, rotated rx -180 ry 0 rz -88.32 deg; joints [25.988, 17.43, -8.212, 41.857, -29.472, -58.291]
  Set speed (5.6 mm/s)
  MoveL 2321 to (922.45, 2304.8, 533.29) mm, rotated rx -180 ry 0 rz -88.32 deg; joints [25.988, 17.783, -8.613, 42.766, -28.915, -59.332]
  MoveL 2322 to (922.45, 2304.8, 513.19) mm, rotated rx -180 ry 0 rz -88.32 deg; joints [25.988, 18.103, -8.951, 43.588, -28.435, -60.27]
  Set speed (91.9 mm/s)
  MoveL 2323 to (923.05, 2373.37, 513.19) mm, rotated rx -180 ry 0 rz -88.32 deg; joints [25.219, 21.008, -5.331, 42.107, -28.492, -58.192]
  MoveL 2324 to (923.16, 2386.07, 513.19) mm, rotated rx 180 ry 0 rz -88.32 deg; joints [25.081, 21.55, -4.645, 41.822, -28.516, -57.797]
  Set speed (100.0 mm/s)
  MoveL 2325 to (923.16, 2386.07, 556.29) mm, rotated rx -180 ry 0 rz -88.32 deg; joints [25.081, 20.906, -3.904, 40.185, -29.561, -55.926]
  MoveL 2326 to (1073.03, 2819.74, 556.29) mm, rotated rx -180 ry 0 rz -88.32 deg; joints [24.047, 44.59, 28.856, 31.144, -36.398, -44.75]
  Set speed (5.6 mm/s)
  MoveL 2327 to (1073.03, 2819.74, 552.29) mm, rotated rx 180 ry 0 rz -88.32 deg; joints [24.047, 44.624, 28.768, 31.23, -36.294, -44.856]
  MoveL 2328 to (1073.03, 2819.74, 532.29) mm, rotated rx -180 ry 0 rz -88.32 deg; joints [24.047, 44.799, 28.335, 31.666, -35.775, -45.396]
  Set speed (91.9 mm/s)
  MoveL 2329 to (752.63, 2822.56, 532.29) mm, rotated rx -180 ry 0 rz -88.32 deg; joints [17.442, 38.455, 19.012, 27.526, -30.074, -38.046]
  Set speed (100.0 mm/s)
  MoveL 2330 to (752.63, 2822.56, 556.29) mm, rotated rx -180 ry 0 rz -88.32 deg; joints [17.442, 38.197, 19.482, 26.958, -30.721, -37.388]
  MoveL 2331 to (752.12, 2822.57, 556.29) mm, rotated rx -180 ry 0 rz -88.32 deg; joints [17.431, 38.189, 19.471, 26.948, -30.713, -37.373]
  Set speed (5.6 mm/s)
  MoveL 2332 to (752.12, 2822.57, 552.29) mm, rotated rx -180 ry 0 rz -88.32 deg; joints [17.431, 38.231, 19.391, 27.041, -30.605, -37.481]
  MoveL 2333 to (752.12, 2822.57, 532.29) mm, rotated rx -180 ry 0 rz -88.32 deg; joints [17.431, 38.447, 19, 27.516, -30.066, -38.031]
  Set speed (91.9 mm/s)
  MoveL 2334 to (736.5, 2822.7, 532.29) mm, rotated rx -180 ry 0 rz -88.32 deg; joints [17.095, 38.203, 18.649, 27.226, -29.825, -37.567]
  Set speed (100.0 mm/s)
  MoveL 2335 to (736.5, 2822.7, 556.29) mm, rotated rx 180 ry 0 rz -88.32 deg; joints [17.095, 37.943, 19.117, 26.658, -30.474, -36.91]
  MoveL 2336 to (758.67, 2816.16, 556.29) mm, rotated rx -180 ry 0 rz -88.32 deg; joints [17.615, 37.964, 19.146, 27.225, -30.705, -37.764]
  Set speed (5.6 mm/s)
  MoveL 2337 to (758.67, 2816.16, 552.29) mm, rotated rx -180 ry 0 rz -88.32 deg; joints [17.615, 38.006, 19.067, 27.319, -30.596, -37.873]
  MoveL 2338 to (758.67, 2816.16, 532.29) mm, rotated rx -180 ry 0 rz -88.32 deg; joints [17.615, 38.223, 18.677, 27.799, -30.059, -38.429]
  Set speed (91.9 mm/s)
  MoveL 2339 to (757.98, 2737.88, 532.29) mm, rotated rx -180 ry 0 rz -88.32 deg; joints [18.148, 34.283, 13.077, 29.806, -28.844, -40.947]
  Set speed (100.0 mm/s)
  MoveL 2340 to (757.98, 2737.88, 556.29) mm, rotated rx -180 ry 0 rz -88.32 deg; joints [18.148, 33.999, 13.526, 29.16, -29.482, -40.207]
  MoveL 2341 to (758.67, 2816.16, 556.29) mm, rotated rx -180 ry 0 rz -88.32 deg; joints [17.615, 37.964, 19.146, 27.225, -30.705, -37.764]
  Set speed (5.6 mm/s)
  MoveL 2342 to (758.67, 2816.16, 533.29) mm, rotated rx -180 ry 0 rz -88.32 deg; joints [17.615, 38.212, 18.697, 27.775, -30.086, -38.401]
  MoveL 2343 to (758.67, 2816.16, 513.19) mm, rotated rx -180 ry 0 rz -88.32 deg; joints [17.615, 38.44, 18.319, 28.271, -29.551, -38.973]
  Set speed (91.9 mm/s)
  MoveL 2344 to (757.98, 2737.88, 513.19) mm, rotated rx 180 ry 0 rz -88.32 deg; joints [18.148, 34.52, 12.734, 30.34, -28.342, -41.554]
  Set speed (100.0 mm/s)
  MoveL 2345 to (757.98, 2737.88, 556.29) mm, rotated rx -180 ry 0 rz -88.32 deg; joints [18.148, 33.999, 13.526, 29.16, -29.482, -40.207]
  MoveL 2346 to (1073.03, 2819.74, 556.29) mm, rotated rx -180 ry 0 rz -88.32 deg; joints [24.047, 44.59, 28.856, 31.144, -36.398, -44.75]
  Set speed (5.6 mm/s)
  MoveL 2347 to (1073.03, 2819.74, 533.29) mm, rotated rx -180 ry 0 rz -88.32 deg; joints [24.047, 44.79, 28.357, 31.644, -35.801, -45.368]
  MoveL 2348 to (1073.03, 2819.74, 513.19) mm, rotated rx -180 ry 0 rz -88.32 deg; joints [24.047, 44.978, 27.939, 32.092, -35.286, -45.919]
  Set speed (91.9 mm/s)
  MoveL 2349 to (752.63, 2822.56, 513.19) mm, rotated rx -180 ry 0 rz -88.32 deg; joints [17.442, 38.671, 18.653, 27.993, -29.565, -38.585]
  Set speed (100.0 mm/s)
  MoveL 2350 to (752.63, 2822.56, 556.29) mm, rotated rx -180 ry 0 rz -88.32 deg; joints [17.442, 38.197, 19.482, 26.958, -30.721, -37.388]
  MoveL 2351 to (723.14, 2747.89, 556.29) mm, rotated rx -180 ry 0 rz -88.32 deg; joints [17.309, 33.943, 13.447, 28.243, -29.085, -38.82]
  Set speed (5.6 mm/s)
  MoveL 2352 to (723.14, 2747.89, 552.29) mm, rotated rx -180 ry 0 rz -88.32 deg; joints [17.309, 33.989, 13.371, 28.348, -28.977, -38.939]
  MoveL 2353 to (723.14, 2747.89, 532.29) mm, rotated rx -180 ry 0 rz -88.32 deg; joints [17.309, 34.227, 12.999, 28.882, -28.441, -39.548]
  Set speed (91.9 mm/s)
  MoveL 2354 to (723.75, 2816.47, 532.29) mm, rotated rx 180 ry 0 rz -88.32 deg; joints [16.862, 37.68, 17.898, 27.144, -29.521, -37.383]
  MoveL 2355 to (723.86, 2829.17, 532.29) mm, rotated rx 180 ry 0 rz -88.32 deg; joints [16.781, 38.338, 18.843, 26.823, -29.743, -36.982]
  Set speed (100.0 mm/s)
  MoveL 2356 to (723.86, 2829.17, 556.29) mm, rotated rx 180 ry 0 rz -88.32 deg; joints [16.781, 38.08, 19.313, 26.261, -30.395, -36.333]
  MoveL 2357 to (752.12, 2822.57, 556.29) mm, rotated rx -180 ry 0 rz -88.32 deg; joints [17.431, 38.189, 19.471, 26.948, -30.713, -37.373]
  Set speed (5.6 mm/s)
  MoveL 2358 to (752.12, 2822.57, 533.29) mm, rotated rx -180 ry 0 rz -88.32 deg; joints [17.431, 38.436, 19.019, 27.492, -30.093, -38.003]
  MoveL 2359 to (752.12, 2822.57, 513.19) mm, rotated rx -180 ry 0 rz -88.32 deg; joints [17.431, 38.663, 18.641, 27.984, -29.557, -38.57]
  Set speed (91.9 mm/s)
  MoveL 2360 to (736.5, 2822.7, 513.19) mm, rotated rx -180 ry 0 rz -88.32 deg; joints [17.095, 38.42, 18.29, 27.694, -29.314, -38.105]
  Set speed (100.0 mm/s)
  MoveL 2361 to (736.5, 2822.7, 556.29) mm, rotated rx 180 ry 0 rz -88.32 deg; joints [17.095, 37.943, 19.117, 26.658, -30.474, -36.91]
  MoveL 2362 to (723.14, 2747.89, 556.29) mm, rotated rx -180 ry 0 rz -88.32 deg; joints [17.309, 33.943, 13.447, 28.243, -29.085, -38.82]
  Set speed (5.6 mm/s)
  MoveL 2363 to (723.14, 2747.89, 533.29) mm, rotated rx -180 ry 0 rz -88.32 deg; joints [17.309, 34.215, 13.017, 28.855, -28.468, -39.517]
  MoveL 2364 to (723.14, 2747.89, 513.19) mm, rotated rx -180 ry 0 rz -88.32 deg; joints [17.309, 34.464, 12.656, 29.409, -27.935, -40.146]
  Set speed (91.9 mm/s)
  MoveL 2365 to (723.75, 2816.47, 513.19) mm, rotated rx -180 ry 0 rz -88.32 deg; joints [16.862, 37.9, 17.542, 27.617, -29.01, -37.924]
  MoveL 2366 to (723.86, 2829.17, 513.19) mm, rotated rx -180 ry 0 rz -88.32 deg; joints [16.781, 38.554, 18.485, 27.286, -29.231, -37.514]
  Set speed (100.0 mm/s)
  MoveL 2367 to (723.86, 2829.17, 566.29) mm, rotated rx -180 ry 0 rz -88.32 deg; joints [16.781, 37.976, 19.515, 26.033, -30.669, -36.068]
  MoveL 2368 to (723.86, 2829.17, 566.29) mm, rotated rx -180 ry 0 rz -88.32 deg; joints [16.781, 37.976, 19.515, 26.033, -30.669, -36.068]
  MoveL 2369 to (723.86, 2829.17, 666.29) mm, rotated rx 180 ry 0 rz -88.32 deg; joints [16.781, 37.099, 21.743, 23.94, -33.484, -33.598]

--- program Blade_handles_west (robot Kawasaki BX130X) ---
  Smooth(1)
  Print: /'Front wall cutout v12'
  Print: /''
  Print: /'Blade handles West'
  Set speed (100.0 mm/s)
  Set Ref.: Work hold down
  Set Tool: Sawblade
  Show Sawblade
  MoveJ 1 to (1013.34, 1635.95, 666.29) mm, rotated rx 180 ry 0 rz -90.5 deg; joints [37.029, -13.288, -32.809, 41.963, -40.111, -63.595]
  MoveL 2 to (1013.34, 1635.95, 666.29) mm, rotated rx 180 ry 0 rz -90.5 deg; joints [37.029, -13.288, -32.809, 41.963, -40.111, -63.595]
  MoveL 3 to (1013.34, 1635.95, 566.29) mm, rotated rx 180 ry 0 rz -90.5 deg; joints [37.029, -12.008, -35.267, 45.173, -37.401, -67.71]
  MoveL 4 to (1013.34, 1635.95, 566.29) mm, rotated rx 180 ry 0 rz -90.5 deg; joints [37.029, -12.008, -35.267, 45.173, -37.401, -67.71]
  Set speed (100.0 mm/s)
  MoveL 5 to (1013.34, 1635.95, 556.29) mm, rotated rx 180 ry 0 rz -90.5 deg; joints [37.029, -11.859, -35.497, 45.528, -37.135, -68.156]
  Set speed (5.6 mm/s)
  MoveL 6 to (1013.34, 1635.95, 551.89) mm, rotated rx 180 ry 0 rz -90.5 deg; joints [37.029, -11.792, -35.598, 45.686, -37.018, -68.354]
  MoveL 7 to (1013.34, 1635.95, 513.19) mm, rotated rx 180 ry 0 rz -90.5 deg; joints [37.029, -11.173, -36.457, 47.133, -35.998, -70.154]
  Set speed (133.3 mm/s)
  MoveL 8 to (1013.78, 1686.75, 513.19) mm, rotated rx -180 ry 0 rz -90.5 deg; joints [35.949, -8.99, -34.553, 46.948, -35.088, -69.352]
  MoveL 9 to (1017.48, 2106.73, 513.19) mm, rotated rx 180 ry 0 rz -90.5 deg; joints [28.824, 8.743, -16.848, 42.992, -30.517, -60.994]
  Set speed (100.0 mm/s)
  MoveL 10 to (1017.48, 2106.73, 566.29) mm, rotated rx -180 ry 0 rz -90.5 deg; joints [28.824, 7.979, -15.786, 40.974, -31.874, -58.635]
  MoveL 11 to (1017.48, 2106.73, 566.29) mm, rotated rx -180 ry 0 rz -90.5 deg; joints [28.824, 7.979, -15.786, 40.974, -31.874, -58.635]
  MoveL 12 to (1017.48, 2106.73, 666.29) mm, rotated rx 180 ry 0 rz -90.5 deg; joints [28.824, 6.766, -13.563, 37.648, -34.534, -54.661]
  Print: /'Blade handles East'

--- program Blade_handles_east (robot Kawasaki BX130X) ---
  Smooth(1)
  Set speed (100.0 mm/s)
  Set Ref.: Work hold down
  Set Tool: Sawblade
  Show Sawblade
  MoveJ 1 to (950.37, 1699.88, 666.29) mm, rotated rx 180 ry 0 rz -90.5 deg; joints [33.808, -12.459, -32.112, 40.328, -38.009, -60.096]
  MoveL 2 to (950.37, 1699.88, 666.29) mm, rotated rx 180 ry 0 rz -90.5 deg; joints [33.808, -12.459, -32.112, 40.328, -38.009, -60.096]
  MoveL 3 to (950.37, 1699.88, 566.29) mm, rotated rx -180 ry 0 rz -90.5 deg; joints [33.808, -11.175, -34.555, 43.685, -35.238, -64.277]
  MoveL 4 to (950.37, 1699.88, 566.29) mm, rotated rx -180 ry 0 rz -90.5 deg; joints [33.808, -11.175, -34.555, 43.685, -35.238, -64.277]
  Set speed (100.0 mm/s)
  MoveL 5 to (950.37, 1699.88, 556.29) mm, rotated rx -180 ry 0 rz -90.5 deg; joints [33.808, -11.026, -34.784, 44.058, -34.966, -64.733]
  Set speed (5.6 mm/s)
  MoveL 6 to (950.37, 1699.88, 551.89) mm, rotated rx 180 ry 0 rz -90.5 deg; joints [33.808, -10.959, -34.884, 44.224, -34.846, -64.935]
  MoveL 7 to (950.37, 1699.88, 513.19) mm, rotated rx 180 ry 0 rz -90.5 deg; joints [33.808, -10.339, -35.737, 45.749, -33.804, -66.782]
  Set speed (133.3 mm/s)
  MoveL 8 to (951.49, 1827.11, 513.19) mm, rotated rx 180 ry 0 rz -90.5 deg; joints [31.437, -4.73, -30.665, 45.045, -31.905, -64.722]
  MoveL 9 to (954.4, 2157.1, 513.19) mm, rotated rx 180 ry 0 rz -90.5 deg; joints [26.52, 9.472, -16.035, 41.199, -29.185, -57.781]
  Set speed (100.0 mm/s)
  MoveL 10 to (954.4, 2157.1, 566.29) mm, rotated rx -180 ry 0 rz -90.5 deg; joints [26.52, 8.713, -14.974, 39.156, -30.575, -55.425]
  MoveL 11 to (954.4, 2157.1, 566.29) mm, rotated rx -180 ry 0 rz -90.5 deg; joints [26.52, 8.713, -14.974, 39.156, -30.575, -55.425]
  MoveL 12 to (954.4, 2157.1, 666.29) mm, rotated rx 180 ry 0 rz -90.5 deg; joints [26.52, 7.509, -12.755, 35.812, -33.294, -51.486]
  Print: /'Handles roughing'

--- program Handles_roughing (robot Kawasaki BX130X) ---
  Smooth(1)
  Set speed (100.0 mm/s)
  Set Ref.: Work hold down
  Set Tool: halfInchUpcut
  Show halfInchUpcut
  MoveJ 1 to (1013.58, 1832.8, 666.29) mm, rotated rx -180 ry 0 rz -77.47 deg; joints [37.043, 0.991, -22.608, 49.213, -45.308, -78.876]
  MoveL 2 to (1013.58, 1832.8, 666.29) mm, rotated rx -180 ry 0 rz -77.47 deg; joints [37.043, 0.991, -22.608, 49.213, -45.308, -78.876]
  MoveL 3 to (1013.58, 1832.8, 566.29) mm, rotated rx -180 ry 0 rz -77.47 deg; joints [37.043, 2.529, -24.64, 52.056, -43.041, -82.839]
  MoveL 4 to (1013.58, 1832.8, 566.29) mm, rotated rx -180 ry 0 rz -77.47 deg; joints [37.043, 2.529, -24.64, 52.056, -43.041, -82.839]
  Set speed (100.0 mm/s)
  MoveL 5 to (1013.58, 1832.8, 556.29) mm, rotated rx -180 ry 0 rz -77.47 deg; joints [37.043, 2.701, -24.828, 52.361, -42.822, -83.255]
  Set speed (5.6 mm/s)
  MoveL 6 to (1013.58, 1832.8, 552.29) mm, rotated rx -180 ry 0 rz -77.47 deg; joints [37.043, 2.77, -24.902, 52.484, -42.734, -83.423]
  MoveL 7 to (1013.58, 1832.8, 531.29) mm, rotated rx -180 ry 0 rz -77.47 deg; joints [37.043, 3.144, -25.283, 53.14, -42.278, -84.313]
  Set speed (91.9 mm/s)
  MoveL 8 to (999.6, 1832.92, 531.29) mm, rotated rx -180 ry 0 rz -77.47 deg; joints [36.689, 2.742, -25.701, 53.115, -42.019, -84.052]
  MoveL 9 to (999.6, 1832.92, 531.29) mm, rotated rx -180 ry 0 rz -77.47 deg; joints [36.689, 2.742, -25.701, 53.115, -42.019, -84.052]
  MoveC 10 to (991.49, 1829.64, 531.29) mm, rotated rx -180 ry 0 rz -77.47 deg; joints [36.545, 2.379, -26.076, 53.11, -41.911, -83.953] to (988.07, 1821.59, 531.29) mm, rotated rx 180 ry 0 rz -77.47 deg; joints [36.61, 1.964, -26.502, 53.128, -41.95, -84.019]
  MoveL 11 to (987.04, 1704.76, 531.29) mm, rotated rx -180 ry 0 rz -77.47 deg; joints [38.922, -2.641, -31.087, 53.324, -43.59, -85.786]
  MoveL 12 to (987.04, 1704.76, 531.29) mm, rotated rx -180 ry 0 rz -77.47 deg; joints [38.922, -2.641, -31.087, 53.324, -43.59, -85.786]
  MoveC 13 to (990.32, 1696.65, 531.29) mm, rotated rx 180 ry 0 rz -77.47 deg; joints [39.179, -2.855, -31.293, 53.337, -43.776, -85.973] to (998.37, 1693.23, 531.29) mm, rotated rx -180 ry 0 rz -77.47 deg; joints [39.461, -2.731, -31.174, 53.36, -43.972, -86.192]
  MoveL 14 to (1012.33, 1693.11, 531.29) mm, rotated rx -180 ry 0 rz -77.47 deg; joints [39.824, -2.288, -30.745, 53.396, -44.22, -86.482]
  Set speed (100.0 mm/s)
  MoveL 15 to (1012.33, 1693.11, 556.29) mm, rotated rx 180 ry 0 rz -77.47 deg; joints [39.824, -2.746, -30.273, 52.639, -44.779, -85.422]
  MoveL 16 to (1011.78, 1629.61, 556.29) mm, rotated rx -180 ry 0 rz -77.47 deg; joints [41.209, -5.215, -32.616, 52.639, -45.833, -86.33]
  Set speed (5.6 mm/s)
  MoveL 17 to (1011.78, 1629.61, 552.29) mm, rotated rx -180 ry 0 rz -77.47 deg; joints [41.209, -5.143, -32.694, 52.756, -45.741, -86.497]
  MoveL 18 to (1011.78, 1629.61, 531.29) mm, rotated rx -180 ry 0 rz -77.47 deg; joints [41.209, -4.751, -33.096, 53.379, -45.265, -87.386]
  Set speed (91.9 mm/s)
  MoveL 19 to (987.65, 1629.82, 531.29) mm, rotated rx -180 ry 0 rz -77.47 deg; joints [40.574, -5.554, -33.845, 53.304, -44.848, -86.854]
  MoveL 20 to (987.65, 1629.82, 531.29) mm, rotated rx -180 ry 0 rz -77.47 deg; joints [40.574, -5.554, -33.845, 53.304, -44.848, -86.854]
  MoveC 21 to (976.91, 1634.38, 531.29) mm, rotated rx -180 ry 0 rz -77.47 deg; joints [40.187, -5.733, -34.012, 53.271, -44.582, -86.549] to (972.55, 1645.2, 531.29) mm, rotated rx 180 ry 0 rz -77.47 deg; joints [39.829, -5.451, -33.75, 53.265, -44.318, -86.304]
  MoveL 22 to (972.6, 1651.55, 531.29) mm, rotated rx -180 ry 0 rz -77.47 deg; joints [39.69, -5.198, -33.515, 53.271, -44.209, -86.219]
  MoveC 23 to (967.91, 1669.86, 531.29) mm, rotated rx -180 ry 0 rz -77.47 deg; joints [39.164, -4.626, -32.979, 53.264, -43.816, -85.862] to (954.75, 1683.44, 531.29) mm, rotated rx 180 ry 0 rz -77.47 deg; joints [38.52, -4.508, -32.868, 53.219, -43.358, -85.378]
  MoveC 24 to (947.95, 1690.45, 531.29) mm, rotated rx 180 ry 0 rz -77.47 deg; joints [38.187, -4.443, -32.806, 53.194, -43.121, -85.127] to (945.52, 1699.92, 531.29) mm, rotated rx -180 ry 0 rz -77.47 deg; joints [37.922, -4.139, -32.519, 53.185, -42.924, -84.942]
  Set speed (100.0 mm/s)
  MoveL 25 to (945.52, 1699.92, 556.29) mm, rotated rx -180 ry 0 rz -77.47 deg; joints [37.922, -4.602, -32.041, 52.387, -43.494, -83.847]
  MoveL 26 to (1011.78, 1629.61, 556.29) mm, rotated rx -180 ry 0 rz -77.47 deg; joints [41.209, -5.215, -32.616, 52.639, -45.833, -86.33]
  Set speed (5.6 mm/s)
  MoveL 27 to (1011.78, 1629.61, 532.29) mm, rotated rx -180 ry 0 rz -77.47 deg; joints [41.209, -4.77, -33.077, 53.349, -45.287, -87.344]
  MoveL 28 to (1011.78, 1629.61, 513.19) mm, rotated rx -180 ry 0 rz -77.47 deg; joints [41.209, -4.401, -33.432, 53.931, -44.858, -88.168]
  Set speed (91.9 mm/s)
  MoveL 29 to (987.65, 1629.82, 513.19) mm, rotated rx -180 ry 0 rz -77.47 deg; joints [40.574, -5.202, -34.183, 53.867, -44.438, -87.644]
  MoveL 30 to (987.65, 1629.82, 513.19) mm, rotated rx 180 ry 0 rz -77.47 deg; joints [40.574, -5.202, -34.183, 53.867, -44.438, -87.644]
  MoveC 31 to (976.91, 1634.38, 513.19) mm, rotated rx 180 ry 0 rz -77.47 deg; joints [40.187, -5.381, -34.35, 53.839, -44.172, -87.344] to (972.55, 1645.2, 513.19) mm, rotated rx -180 ry 0 rz -77.47 deg; joints [39.829, -5.099, -34.088, 53.838, -43.908, -87.1]
  MoveL 32 to (972.6, 1651.55, 513.19) mm, rotated rx -180 ry 0 rz -77.47 deg; joints [39.69, -4.847, -33.852, 53.844, -43.8, -87.016]
  MoveC 33 to (967.91, 1669.86, 513.19) mm, rotated rx -180 ry 0 rz -77.47 deg; joints [39.164, -4.276, -33.315, 53.843, -43.409, -86.662] to (954.75, 1683.44, 513.19) mm, rotated rx -180 ry 0 rz -77.47 deg; joints [38.52, -4.158, -33.203, 53.807, -42.95, -86.184]
  MoveC 34 to (947.95, 1690.45, 513.19) mm, rotated rx -180 ry 0 rz -77.47 deg; joints [38.187, -4.093, -33.141, 53.786, -42.714, -85.936] to (945.52, 1699.92, 513.19) mm, rotated rx 180 ry 0 rz -77.47 deg; joints [37.922, -3.79, -32.854, 53.78, -42.518, -85.752]
  Set speed (100.0 mm/s)
  MoveL 35 to (945.52, 1699.92, 556.29) mm, rotated rx -180 ry 0 rz -77.47 deg; joints [37.922, -4.602, -32.041, 52.387, -43.494, -83.847]
  MoveL 36 to (946.64, 1827.15, 556.29) mm, rotated rx -180 ry 0 rz -77.47 deg; joints [35.433, 0.542, -27.032, 52.183, -41.665, -82.008]
  Set speed (5.6 mm/s)
  MoveL 37 to (946.64, 1827.15, 552.29) mm, rotated rx -180 ry 0 rz -77.47 deg; joints [35.433, 0.613, -27.107, 52.312, -41.575, -82.182]
  MoveL 38 to (946.64, 1827.15, 531.29) mm, rotated rx -180 ry 0 rz -77.47 deg; joints [35.433, 0.992, -27.493, 53.004, -41.111, -83.103]
  Set speed (91.9 mm/s)
  MoveC 39 to (949.23, 1836.59, 531.29) mm, rotated rx -180 ry 0 rz -77.47 deg; joints [35.325, 1.442, -27.036, 52.983, -41.04, -83.008] to (956.16, 1843.49, 531.29) mm, rotated rx 180 ry 0 rz -77.47 deg; joints [35.378, 1.913, -26.554, 52.981, -41.083, -83.038]
  MoveC 40 to (969.56, 1856.83, 531.29) mm, rotated rx -180 ry 0 rz -77.47 deg; joints [35.479, 2.821, -25.619, 52.969, -41.171, -83.085] to (974.57, 1875.06, 531.29) mm, rotated rx -180 ry 0 rz -77.47 deg; joints [35.276, 3.681, -24.722, 52.909, -41.05, -82.878]
  MoveL 41 to (974.63, 1881.41, 531.29) mm, rotated rx -180 ry 0 rz -77.47 deg; joints [35.164, 3.933, -24.458, 52.882, -40.979, -82.772]
  MoveL 42 to (974.63, 1881.41, 531.29) mm, rotated rx -180 ry 0 rz -77.47 deg; joints [35.164, 3.933, -24.458, 52.882, -40.979, -82.772]
  MoveC 43 to (979.19, 1892.14, 531.29) mm, rotated rx 180 ry 0 rz -77.47 deg; joints [35.088, 4.483, -23.878, 52.844, -40.944, -82.674] to (990, 1896.51, 531.29) mm, rotated rx -180 ry 0 rz -77.47 deg; joints [35.283, 4.954, -23.378, 52.844, -41.098, -82.797]
  MoveL 44 to (1014.13, 1896.3, 531.29) mm, rotated rx -180 ry 0 rz -77.47 deg; joints [35.888, 5.619, -22.667, 52.882, -41.55, -83.229]
  Set speed (100.0 mm/s)
  MoveL 45 to (1014.13, 1896.3, 556.29) mm, rotated rx 180 ry 0 rz -77.47 deg; joints [35.888, 5.185, -22.217, 52.098, -42.089, -82.177]
  MoveL 46 to (1021.09, 1965.98, 556.29) mm, rotated rx 180 ry 0 rz -77.47 deg; joints [34.846, 8.093, -19.062, 51.718, -41.513, -81.027]
  Set speed (5.6 mm/s)
  MoveL 47 to (1021.09, 1965.98, 552.29) mm, rotated rx -180 ry 0 rz -77.47 deg; joints [34.846, 8.159, -19.134, 51.842, -41.427, -81.192]
  MoveL 48 to (1021.09, 1965.98, 531.29) mm, rotated rx 180 ry 0 rz -77.47 deg; joints [34.846, 8.516, -19.506, 52.499, -40.98, -82.066]
  Set speed (91.9 mm/s)
  MoveC 49 to (1018.5, 1956.55, 531.29) mm, rotated rx -180 ry 0 rz -77.47 deg; joints [34.943, 8.08, -19.989, 52.556, -41.019, -82.202] to (1011.58, 1949.64, 531.29) mm, rotated rx 180 ry 0 rz -77.47 deg; joints [34.892, 7.623, -20.493, 52.591, -40.955, -82.216]
  MoveL 50 to (1011.57, 1949.64, 531.29) mm, rotated rx -180 ry 0 rz -77.47 deg; joints [34.892, 7.623, -20.493, 52.591, -40.955, -82.216]
  MoveC 51 to (998.18, 1936.3, 531.29) mm, rotated rx -180 ry 0 rz -77.47 deg; joints [34.791, 6.738, -21.46, 52.652, -40.834, -82.233] to (993.16, 1918.07, 531.29) mm, rotated rx -180 ry 0 rz -77.47 deg; joints [34.982, 5.887, -22.38, 52.743, -40.926, -82.473]
  MoveL 52 to (993.11, 1911.72, 531.29) mm, rotated rx -180 ry 0 rz -77.47 deg; joints [35.092, 5.636, -22.649, 52.775, -40.992, -82.585]
  MoveL 53 to (993.11, 1911.72, 531.29) mm, rotated rx -180 ry 0 rz -77.47 deg; joints [35.092, 5.636, -22.649, 52.775, -40.992, -82.585]
  MoveC 54 to (988.55, 1900.99, 531.29) mm, rotated rx -180 ry 0 rz -77.47 deg; joints [35.167, 5.09, -23.234, 52.821, -41.022, -82.692] to (977.73, 1896.62, 531.29) mm, rotated rx -180 ry 0 rz -77.47 deg; joints [34.971, 4.619, -23.734, 52.821, -40.867, -82.569]
  MoveL 55 to (953.6, 1896.83, 531.29) mm, rotated rx -180 ry 0 rz -77.47 deg; joints [34.352, 3.966, -24.423, 52.765, -40.411, -82.108]
  Set speed (100.0 mm/s)
  MoveL 56 to (953.6, 1896.83, 556.29) mm, rotated rx 180 ry 0 rz -77.47 deg; joints [34.352, 3.526, -23.969, 51.942, -40.957, -81.023]
  MoveL 57 to (954.16, 1960.33, 556.29) mm, rotated rx 180 ry 0 rz -77.47 deg; joints [33.282, 6.081, -21.257, 51.605, -40.309, -79.93]
  Set speed (5.6 mm/s)
  MoveL 58 to (954.16, 1960.33, 552.29) mm, rotated rx -180 ry 0 rz -77.47 deg; joints [33.282, 6.149, -21.329, 51.735, -40.221, -80.1]
  MoveL 59 to (954.16, 1960.33, 531.29) mm, rotated rx -180 ry 0 rz -77.47 deg; joints [33.282, 6.512, -21.704, 52.429, -39.768, -81.007]
  Set speed (91.9 mm/s)
  MoveL 60 to (968.13, 1960.21, 531.29) mm, rotated rx -180 ry 0 rz -77.47 deg; joints [33.636, 6.875, -21.311, 52.46, -40.034, -81.264]
  MoveL 61 to (968.13, 1960.21, 531.29) mm, rotated rx -180 ry 0 rz -77.47 deg; joints [33.636, 6.875, -21.311, 52.46, -40.034, -81.264]
  MoveC 62 to (976.24, 1963.49, 531.29) mm, rotated rx 180 ry 0 rz -77.47 deg; joints [33.784, 7.219, -20.935, 52.455, -40.157, -81.349] to (979.66, 1971.54, 531.29) mm, rotated rx -180 ry 0 rz -77.47 deg; joints [33.736, 7.627, -20.488, 52.41, -40.146, -81.26]
  MoveL 63 to (980.69, 2088.37, 531.29) mm, rotated rx -180 ry 0 rz -77.47 deg; joints [31.916, 12.285, -15.234, 51.499, -39.246, -78.973]
  MoveL 64 to (980.69, 2088.37, 531.29) mm, rotated rx -180 ry 0 rz -77.47 deg; joints [31.916, 12.285, -15.234, 51.499, -39.246, -78.973]
  MoveC 65 to (977.42, 2096.48, 531.29) mm, rotated rx -180 ry 0 rz -77.47 deg; joints [31.716, 12.527, -14.953, 51.418, -39.131, -78.75] to (969.36, 2099.9, 531.29) mm, rotated rx -180 ry 0 rz -77.47 deg; joints [31.47, 12.466, -15.024, 51.374, -38.955, -78.546]
  MoveL 66 to (955.39, 2100.02, 531.29) mm, rotated rx -180 ry 0 rz -77.47 deg; joints [31.129, 12.13, -15.413, 51.348, -38.686, -78.311]
  Set speed (100.0 mm/s)
  MoveL 67 to (955.39, 2100.02, 556.29) mm, rotated rx 180 ry 0 rz -77.47 deg; joints [31.129, 11.721, -14.974, 50.533, -39.22, -77.264]
  MoveL 68 to (955.95, 2163.52, 556.29) mm, rotated rx -180 ry 0 rz -77.47 deg; joints [30.233, 14.304, -11.964, 49.895, -38.877, -75.928]
  Set speed (5.6 mm/s)
  MoveL 69 to (955.95, 2163.52, 552.29) mm, rotated rx -180 ry 0 rz -77.47 deg; joints [30.233, 14.367, -12.035, 50.023, -38.791, -76.091]
  MoveL 70 to (955.95, 2163.52, 531.29) mm, rotated rx -180 ry 0 rz -77.47 deg; joints [30.233, 14.702, -12.4, 50.7, -38.344, -76.957]
  Set speed (91.9 mm/s)
  MoveL 71 to (980.08, 2163.31, 531.29) mm, rotated rx -180 ry 0 rz -77.47 deg; joints [30.81, 15.267, -11.728, 50.741, -38.81, -77.345]
  MoveL 72 to (980.08, 2163.31, 531.29) mm, rotated rx 180 ry 0 rz -77.47 deg; joints [30.81, 15.267, -11.728, 50.741, -38.81, -77.345]
  MoveC 73 to (990.82, 2158.75, 531.29) mm, rotated rx -180 ry 0 rz -77.47 deg; joints [31.128, 15.343, -11.637, 50.804, -39.039, -77.612] to (995.19, 2147.93, 531.29) mm, rotated rx -180 ry 0 rz -77.47 deg; joints [31.386, 15.016, -12.027, 50.926, -39.177, -77.919]
  MoveL 74 to (995.13, 2141.58, 531.29) mm, rotated rx -180 ry 0 rz -77.47 deg; joints [31.476, 14.761, -12.33, 50.993, -39.209, -78.059]
  MoveC 75 to (999.82, 2123.27, 531.29) mm, rotated rx -180 ry 0 rz -77.47 deg; joints [31.854, 14.147, -13.058, 51.186, -39.4, -78.531] to (1012.98, 2109.69, 531.29) mm, rotated rx -180 ry 0 rz -77.47 deg; joints [32.366, 13.936, -13.306, 51.332, -39.731, -79.025]
  MoveC 76 to (1019.79, 2102.68, 531.29) mm, rotated rx -180 ry 0 rz -77.47 deg; joints [32.632, 13.83, -13.431, 51.405, -39.904, -79.278] to (1022.22, 2093.21, 531.29) mm, rotated rx -180 ry 0 rz -77.47 deg; joints [32.833, 13.519, -13.797, 51.496, -40.01, -79.517]
  Set speed (100.0 mm/s)
  MoveL 77 to (1022.22, 2093.21, 556.29) mm, rotated rx -180 ry 0 rz -77.47 deg; joints [32.833, 13.116, -13.359, 50.724, -40.538, -78.505]
  MoveL 78 to (955.95, 2163.52, 556.29) mm, rotated rx -180 ry 0 rz -77.47 deg; joints [30.233, 14.304, -11.964, 49.895, -38.877, -75.928]
  Set speed (5.6 mm/s)
  MoveL 79 to (955.95, 2163.52, 532.29) mm, rotated rx -180 ry 0 rz -77.47 deg; joints [30.233, 14.686, -12.383, 50.667, -38.365, -76.915]
  MoveL 80 to (955.95, 2163.52, 513.19) mm, rotated rx 180 ry 0 rz -77.47 deg; joints [30.233, 15.001, -12.705, 51.297, -37.964, -77.716]
  Set speed (91.9 mm/s)
  MoveL 81 to (980.08, 2163.31, 513.19) mm, rotated rx -180 ry 0 rz -77.47 deg; joints [30.81, 15.564, -12.032, 51.326, -38.431, -78.094]
  MoveL 82 to (980.08, 2163.31, 513.19) mm, rotated rx -180 ry 0 rz -77.47 deg; joints [30.81, 15.564, -12.032, 51.326, -38.432, -78.094]
  MoveC 83 to (990.82, 2158.75, 513.19) mm, rotated rx -180 ry 0 rz -77.47 deg; joints [31.128, 15.64, -11.942, 51.385, -38.661, -78.358] to (995.19, 2147.93, 513.19) mm, rotated rx -180 ry 0 rz -77.47 deg; joints [31.386, 15.314, -12.332, 51.506, -38.8, -78.666]
  MoveL 84 to (995.13, 2141.58, 513.19) mm, rotated rx -180 ry 0 rz -77.47 deg; joints [31.476, 15.06, -12.635, 51.574, -38.832, -78.807]
  MoveC 85 to (999.82, 2123.27, 513.19) mm, rotated rx -180 ry 0 rz -77.47 deg; joints [31.854, 14.448, -13.363, 51.767, -39.022, -79.281] to (1012.98, 2109.69, 513.19) mm, rotated rx -180 ry 0 rz -77.47 deg; joints [32.366, 14.237, -13.611, 51.908, -39.355, -79.772]
  MoveC 86 to (1019.79, 2102.68, 513.19) mm, rotated rx 180 ry 0 rz -77.47 deg; joints [32.632, 14.132, -13.736, 51.978, -39.528, -80.024] to (1022.22, 2093.21, 513.19) mm, rotated rx -180 ry 0 rz -77.47 deg; joints [32.833, 13.822, -14.102, 52.069, -39.634, -80.264]
  Set speed (100.0 mm/s)
  MoveL 87 to (1022.22, 2093.21, 556.29) mm, rotated rx -180 ry 0 rz -77.47 deg; joints [32.833, 13.116, -13.359, 50.724, -40.538, -78.505]
  MoveL 88 to (1021.09, 1965.98, 556.29) mm, rotated rx 180 ry 0 rz -77.47 deg; joints [34.846, 8.093, -19.062, 51.718, -41.513, -81.027]
  Set speed (5.6 mm/s)
  MoveL 89 to (1021.09, 1965.98, 532.29) mm, rotated rx 180 ry 0 rz -77.47 deg; joints [34.846, 8.499, -19.489, 52.468, -41.001, -82.024]
  MoveL 90 to (1021.09, 1965.98, 513.19) mm, rotated rx -180 ry 0 rz -77.47 deg; joints [34.846, 8.835, -19.816, 53.079, -40.6, -82.832]
  Set speed (91.9 mm/s)
  MoveC 91 to (1018.5, 1956.55, 513.19) mm, rotated rx 180 ry 0 rz -77.47 deg; joints [34.943, 8.399, -20.3, 53.138, -40.639, -82.97] to (1011.58, 1949.64, 513.19) mm, rotated rx -180 ry 0 rz -77.47 deg; joints [34.892, 7.944, -20.804, 53.176, -40.574, -82.988]
  MoveL 92 to (1011.57, 1949.64, 513.19) mm, rotated rx -180 ry 0 rz -77.47 deg; joints [34.892, 7.943, -20.804, 53.176, -40.574, -82.988]
  MoveC 93 to (998.18, 1936.3, 513.19) mm, rotated rx -180 ry 0 rz -77.47 deg; joints [34.791, 7.061, -21.772, 53.243, -40.451, -83.012] to (993.16, 1918.07, 513.19) mm, rotated rx -180 ry 0 rz -77.47 deg; joints [34.982, 6.213, -22.694, 53.337, -40.542, -83.257]
  MoveL 94 to (993.11, 1911.72, 513.19) mm, rotated rx -180 ry 0 rz -77.47 deg; joints [35.092, 5.963, -22.963, 53.369, -40.607, -83.369]
  MoveL 95 to (993.11, 1911.72, 513.19) mm, rotated rx -180 ry 0 rz -77.47 deg; joints [35.092, 5.963, -22.963, 53.369, -40.607, -83.369]
  MoveC 96 to (988.55, 1900.99, 513.19) mm, rotated rx -180 ry 0 rz -77.47 deg; joints [35.167, 5.418, -23.549, 53.416, -40.636, -83.479] to (977.73, 1896.62, 513.19) mm, rotated rx -180 ry 0 rz -77.47 deg; joints [34.971, 4.949, -24.05, 53.421, -40.48, -83.361]
  MoveL 97 to (953.6, 1896.83, 513.19) mm, rotated rx -180 ry 0 rz -77.47 deg; joints [34.352, 4.298, -24.74, 53.377, -40.022, -82.91]
  Set speed (100.0 mm/s)
  MoveL 98 to (953.6, 1896.83, 556.29) mm, rotated rx 180 ry 0 rz -77.47 deg; joints [34.352, 3.526, -23.969, 51.942, -40.957, -81.023]
  MoveL 99 to (954.16, 1960.33, 556.29) mm, rotated rx 180 ry 0 rz -77.47 deg; joints [33.282, 6.081, -21.257, 51.605, -40.309, -79.93]
  Set speed (5.6 mm/s)
  MoveL 100 to (954.16, 1960.33, 532.29) mm, rotated rx -180 ry 0 rz -77.47 deg; joints [33.282, 6.495, -21.687, 52.396, -39.789, -80.963]
  MoveL 101 to (954.16, 1960.33, 513.19) mm, rotated rx -180 ry 0 rz -77.47 deg; joints [33.282, 6.836, -22.017, 53.043, -39.382, -81.802]
  Set speed (91.9 mm/s)
  MoveL 102 to (968.13, 1960.21, 513.19) mm, rotated rx -180 ry 0 rz -77.47 deg; joints [33.636, 7.198, -21.623, 53.066, -39.649, -82.054]
  MoveL 103 to (968.13, 1960.21, 513.19) mm, rotated rx -180 ry 0 rz -77.47 deg; joints [33.636, 7.198, -21.623, 53.066, -39.649, -82.054]
  MoveC 104 to (976.24, 1963.49, 513.19) mm, rotated rx 180 ry 0 rz -77.47 deg; joints [33.784, 7.541, -21.247, 53.057, -39.773, -82.135] to (979.66, 1971.54, 513.19) mm, rotated rx -180 ry 0 rz -77.47 deg; joints [33.736, 7.948, -20.799, 53.01, -39.763, -82.044]
  MoveL 105 to (980.69, 2088.37, 513.19) mm, rotated rx -180 ry 0 rz -77.47 deg; joints [31.916, 12.591, -15.54, 52.092, -38.867, -79.737]
  MoveL 106 to (980.69, 2088.37, 513.19) mm, rotated rx 180 ry 0 rz -77.47 deg; joints [31.916, 12.591, -15.54, 52.092, -38.867, -79.737]
  MoveC 107 to (977.42, 2096.48, 513.19) mm, rotated rx -180 ry 0 rz -77.47 deg; joints [31.716, 12.833, -15.259, 52.013, -38.752, -79.514] to (969.36, 2099.9, 513.19) mm, rotated rx -180 ry 0 rz -77.47 deg; joints [31.47, 12.772, -15.33, 51.972, -38.575, -79.314]
  MoveL 108 to (955.39, 2100.02, 513.19) mm, rotated rx 180 ry 0 rz -77.47 deg; joints [31.129, 12.437, -15.719, 51.953, -38.305, -79.084]
  Set speed (100.0 mm/s)
  MoveL 109 to (955.39, 2100.02, 556.29) mm, rotated rx 180 ry 0 rz -77.47 deg; joints [31.129, 11.721, -14.974, 50.533, -39.22, -77.264]
  MoveL 110 to (946.64, 1827.15, 556.29) mm, rotated rx -180 ry 0 rz -77.47 deg; joints [35.433, 0.542, -27.032, 52.183, -41.665, -82.008]
  Set speed (5.6 mm/s)
  MoveL 111 to (946.64, 1827.15, 532.29) mm, rotated rx -180 ry 0 rz -77.47 deg; joints [35.433, 0.973, -27.475, 52.971, -41.133, -83.059]
  MoveL 112 to (946.64, 1827.15, 513.19) mm, rotated rx -180 ry 0 rz -77.47 deg; joints [35.433, 1.33, -27.816, 53.616, -40.716, -83.913]
  Set speed (91.9 mm/s)
  MoveC 113 to (949.23, 1836.59, 513.19) mm, rotated rx -180 ry 0 rz -77.47 deg; joints [35.325, 1.78, -27.357, 53.595, -40.646, -83.816] to (956.16, 1843.49, 513.19) mm, rotated rx -180 ry 0 rz -77.47 deg; joints [35.378, 2.25, -26.875, 53.589, -40.69, -83.843]
  MoveC 114 to (969.56, 1856.83, 513.19) mm, rotated rx -180 ry 0 rz -77.47 deg; joints [35.479, 3.155, -25.938, 53.571, -40.78, -83.884] to (974.57, 1875.06, 513.19) mm, rotated rx 180 ry 0 rz -77.47 deg; joints [35.276, 4.013, -25.04, 53.51, -40.661, -83.673]
  MoveL 115 to (974.63, 1881.41, 513.19) mm, rotated rx -180 ry 0 rz -77.47 deg; joints [35.164, 4.264, -24.775, 53.484, -40.59, -83.566]
  MoveL 116 to (974.63, 1881.41, 513.19) mm, rotated rx 180 ry 0 rz -77.47 deg; joints [35.164, 4.265, -24.775, 53.484, -40.59, -83.566]
  MoveC 117 to (979.19, 1892.14, 513.19) mm, rotated rx -180 ry 0 rz -77.47 deg; joints [35.088, 4.813, -24.194, 53.444, -40.556, -83.465] to (990, 1896.51, 513.19) mm, rotated rx -180 ry 0 rz -77.47 deg; joints [35.283, 5.283, -23.693, 53.439, -40.712, -83.583]
  MoveL 118 to (1014.13, 1896.3, 513.19) mm, rotated rx -180 ry 0 rz -77.47 deg; joints [35.888, 5.946, -22.982, 53.465, -41.166, -84.005]
  Set speed (100.0 mm/s)
  MoveL 119 to (1014.13, 1896.3, 556.29) mm, rotated rx 180 ry 0 rz -77.47 deg; joints [35.888, 5.185, -22.217, 52.098, -42.089, -82.177]
  MoveL 120 to (1013.58, 1832.8, 556.29) mm, rotated rx -180 ry 0 rz -77.47 deg; joints [37.043, 2.701, -24.828, 52.361, -42.822, -83.255]
  Set speed (5.6 mm/s)
  MoveL 121 to (1013.58, 1832.8, 532.29) mm, rotated rx -180 ry 0 rz -77.47 deg; joints [37.043, 3.126, -25.266, 53.108, -42.299, -84.27]
  MoveL 122 to (1013.58, 1832.8, 513.19) mm, rotated rx -180 ry 0 rz -77.47 deg; joints [37.043, 3.477, -25.602, 53.719, -41.889, -85.094]
  Set speed (91.9 mm/s)
  MoveL 123 to (999.6, 1832.92, 513.19) mm, rotated rx -180 ry 0 rz -77.47 deg; joints [36.689, 3.076, -26.02, 53.702, -41.63, -84.839]
  MoveL 124 to (999.6, 1832.92, 513.19) mm, rotated rx -180 ry 0 rz -77.47 deg; joints [36.689, 3.076, -26.02, 53.702, -41.63, -84.839]
  MoveC 125 to (991.49, 1829.64, 513.19) mm, rotated rx -180 ry 0 rz -77.47 deg; joints [36.545, 2.714, -26.396, 53.7, -41.52, -84.743] to (988.07, 1821.59, 513.19) mm, rotated rx -180 ry 0 rz -77.47 deg; joints [36.61, 2.3, -26.823, 53.719, -41.558, -84.811]
  MoveL 126 to (987.04, 1704.76, 513.19) mm, rotated rx 180 ry 0 rz -77.47 deg; joints [38.922, -2.295, -31.418, 53.901, -43.188, -86.58]
  MoveL 127 to (987.04, 1704.76, 513.19) mm, rotated rx -180 ry 0 rz -77.47 deg; joints [38.922, -2.295, -31.418, 53.901, -43.188, -86.58]
  MoveC 128 to (990.32, 1696.65, 513.19) mm, rotated rx -180 ry 0 rz -77.47 deg; joints [39.179, -2.508, -31.624, 53.911, -43.373, -86.765] to (998.37, 1693.23, 513.19) mm, rotated rx -180 ry 0 rz -77.47 deg; joints [39.461, -2.384, -31.505, 53.93, -43.571, -86.981]
  MoveL 129 to (1012.33, 1693.11, 513.19) mm, rotated rx -180 ry 0 rz -77.47 deg; joints [39.824, -1.942, -31.075, 53.959, -43.82, -87.266]
  Set speed (100.0 mm/s)
  MoveL 130 to (1012.33, 1693.11, 566.29) mm, rotated rx 180 ry 0 rz -77.47 deg; joints [39.824, -2.924, -30.08, 52.344, -45.005, -85.005]
  MoveL 131 to (1012.33, 1693.11, 566.29) mm, rotated rx 180 ry 0 rz -77.47 deg; joints [39.824, -2.924, -30.08, 52.344, -45.005, -85.005]
  MoveL 132 to (1012.33, 1693.11, 666.29) mm, rotated rx -180 ry 0 rz -77.47 deg; joints [39.824, -4.505, -27.982, 49.599, -47.323, -81.043]

--- program Blade_door_east (robot Kawasaki BX130X) ---
  Smooth(1)
  Set speed (100.0 mm/s)
  Set Ref.: Work hold down
  Set Tool: Sawblade
  Show Sawblade
  MoveJ 1 to (752.06, 1515.37, 666.29) mm, rotated rx -180 ry 0 rz -90.5 deg; joints [31.109, -27.196, -43.324, 35.897, -39.198, -53.368]
  MoveL 2 to (752.06, 1515.37, 666.29) mm, rotated rx -180 ry 0 rz -90.5 deg; joints [31.109, -27.196, -43.324, 35.897, -39.198, -53.368]
  MoveL 3 to (752.06, 1515.37, 566.29) mm, rotated rx 180 ry 0 rz -90.5 deg; joints [31.109, -26.113, -46.08, 38.918, -36.148, -57.182]
  MoveL 4 to (752.06, 1515.37, 566.29) mm, rotated rx 180 ry 0 rz -90.5 deg; joints [31.109, -26.113, -46.08, 38.918, -36.148, -57.182]
  Set speed (100.0 mm/s)
  MoveL 5 to (752.06, 1515.37, 556.29) mm, rotated rx 180 ry 0 rz -90.5 deg; joints [31.109, -25.98, -46.34, 39.26, -35.843, -57.605]
  Set speed (5.6 mm/s)
  MoveL 6 to (752.06, 1515.37, 551.89) mm, rotated rx -180 ry 0 rz -90.5 deg; joints [31.109, -25.92, -46.454, 39.412, -35.708, -57.793]
  MoveL 7 to (752.06, 1515.37, 513.19) mm, rotated rx 180 ry 0 rz -90.5 deg; joints [31.109, -25.351, -47.429, 40.827, -34.527, -59.523]
  Set speed (133.3 mm/s)
  MoveL 8 to (762.78, 2732.45, 513.19) mm, rotated rx 180 ry 0 rz -90.5 deg; joints [16.435, 32.056, 12.278, 25.257, -28.857, -35.163]
  Set speed (100.0 mm/s)
  MoveL 9 to (762.78, 2732.45, 566.29) mm, rotated rx 180 ry 0 rz -90.5 deg; joints [16.435, 31.52, 13.402, 24.038, -30.366, -33.762]
  MoveL 10 to (762.78, 2732.45, 566.29) mm, rotated rx 180 ry 0 rz -90.5 deg; joints [16.435, 31.52, 13.402, 24.038, -30.366, -33.762]
  MoveL 11 to (762.78, 2732.45, 666.29) mm, rotated rx 180 ry 0 rz -90.5 deg; joints [16.435, 30.721, 15.792, 22.028, -33.3, -31.397]

--- program checkTableCalibration (robot Kawasaki BX130X) ---
  Set Ref.: CalibrationFrame
  Set Tool: Tool05inchUpcut at (-1.57, 133.94, 455.3) mm, rotated rx 0 ry 45 rz 90 deg
  MoveJ (Home)*
  MoveJ (SW_disc_corner)*
  MoveJ (Home)*
  MoveJ (NW_disc_corner)*
  MoveJ (Home)*
  MoveJ (NE_disc_corner)*
  MoveJ (Home)*
  MoveJ (SE_disc_corner)*
  MoveJ (Home)*

--- program Blade_doorframe_east (robot Kawasaki BX130X) ---
  Smooth(1)
  Print: /'Front wall cutout v15'
  Print: /''
  Print: /'Blade door cutout east'
  Set speed (100.0 mm/s)
  Set Ref.: Work hold down
  Set Tool: Sawblade
  Show Sawblade
  MoveJ 1 to (707.44, 1515.76, 666.29) mm, rotated rx 180 ry 0 rz -90.5 deg; joints [29.411, -28.532, -44.222, 34.395, -38.617, -50.84]
  MoveL 2 to (707.44, 1515.76, 666.29) mm, rotated rx 180 ry 0 rz -90.5 deg; joints [29.411, -28.532, -44.222, 34.395, -38.617, -50.84]
  MoveL 3 to (707.44, 1515.76, 566.29) mm, rotated rx 180 ry 0 rz -90.5 deg; joints [29.411, -27.484, -47.01, 37.375, -35.507, -54.572]
  MoveL 4 to (707.44, 1515.76, 566.29) mm, rotated rx 180 ry 0 rz -90.5 deg; joints [29.411, -27.484, -47.01, 37.375, -35.507, -54.572]
  Set speed (100.0 mm/s)
  MoveL 5 to (707.44, 1515.76, 556.29) mm, rotated rx -180 ry 0 rz -90.5 deg; joints [29.411, -27.354, -47.274, 37.713, -35.194, -54.987]
  Set speed (5.6 mm/s)
  MoveL 6 to (707.44, 1515.76, 551.89) mm, rotated rx 180 ry 0 rz -90.5 deg; joints [29.411, -27.295, -47.389, 37.865, -35.057, -55.172]
  MoveL 7 to (707.44, 1515.76, 513.19) mm, rotated rx -180 ry 0 rz -90.5 deg; joints [29.411, -26.737, -48.378, 39.271, -33.847, -56.877]
  Set speed (133.3 mm/s)
  MoveL 8 to (718.25, 2742.54, 513.19) mm, rotated rx 180 ry 0 rz -90.5 deg; joints [15.367, 31.928, 12.101, 23.981, -28.394, -33.297]
  Set speed (100.0 mm/s)
  MoveL 9 to (718.25, 2742.54, 566.29) mm, rotated rx 180 ry 0 rz -90.5 deg; joints [15.367, 31.39, 13.224, 22.799, -29.918, -31.944]
  MoveL 10 to (718.25, 2742.54, 566.29) mm, rotated rx 180 ry 0 rz -90.5 deg; joints [15.367, 31.39, 13.224, 22.799, -29.918, -31.944]
  MoveL 11 to (718.25, 2742.54, 666.29) mm, rotated rx 180 ry 0 rz -90.5 deg; joints [15.367, 30.588, 15.611, 20.856, -32.878, -29.669]
  Print: /'Blade door edge east'
